    movel([-0.071523, -1.431037, -2.538408, -0.742944, 1.570796, 1.499273],accel_mss,speed_ms,0,blend_radius_m)
    movel([-0.071633, -1.429838, -2.539341, -0.743210, 1.570796, 1.499163],accel_mss,speed_ms,0,blend_radius_m)
    movel([-0.072441, -1.426473, -2.541948, -0.743968, 1.570796, 1.498355],accel_mss,speed_ms,0,blend_radius_m)
    movel([-0.072913, -1.424072, -2.543798, -0.744519, 1.570796, 1.497883],accel_mss,speed_ms,0,blend_radius_m)
    movel([-0.072968, -1.423023, -2.544604, -0.744762, 1.570796, 1.497829],accel_mss,speed_ms,0,blend_radius_m)
    movel([-0.072889, -1.422073, -2.545332, -0.744984, 1.570796, 1.497908],accel_mss,speed_ms,0,blend_radius_m)
    movel([-0.072695, -1.421230, -2.545977, -0.745182, 1.570796, 1.498101],accel_mss,speed_ms,0,blend_radius_m)
    movel([-0.072401, -1.420498, -2.546536, -0.745355, 1.570796, 1.498395],accel_mss,speed_ms,0,blend_radius_m)
    movel([-0.072027, -1.419881, -2.547006, -0.745502, 1.570796, 1.498770],accel_mss,speed_ms,0,blend_radius_m)
    movel([-0.071586, -1.419384, -2.547385, -0.745620, 1.570796, 1.499210],accel_mss,speed_ms,0,blend_radius_m)
    movel([-0.071096, -1.419012, -2.547668, -0.745709, 1.570796, 1.499700],accel_mss,speed_ms,0,blend_radius_m)
    movel([-0.070575, -1.418770, -2.547852, -0.745766, 1.570796, 1.500221],accel_mss,speed_ms,0,blend_radius_m)
    movel([-0.070039, -1.418663, -2.547934, -0.745792, 1.570796, 1.500757],accel_mss,speed_ms,0,blend_radius_m)
    movel([-0.069506, -1.418695, -2.547909, -0.745784, 1.570796, 1.501291],accel_mss,speed_ms,0,blend_radius_m)
    movel([-0.068990, -1.418869, -2.547777, -0.745743, 1.570796, 1.501806],accel_mss,speed_ms,0,blend_radius_m)
    movel([-0.068509, -1.419192, -2.547531, -0.745666, 1.570796, 1.502287],accel_mss,speed_ms,0,blend_radius_m)
    movel([-0.068083, -1.419668, -2.547169, -0.745552, 1.570796, 1.502713],accel_mss,speed_ms,0,blend_radius_m)
    movel([-0.067726, -1.420299, -2.546687, -0.745402, 1.570796, 1.503070],accel_mss,speed_ms,0,blend_radius_m)
    movel([-0.067456, -1.421092, -2.546082, -0.745215, 1.570796, 1.503341],accel_mss,speed_ms,0,blend_radius_m)
    movel([-0.067286, -1.422046, -2.545352, -0.744991, 1.570796, 1.503511],accel_mss,speed_ms,0,blend_radius_m)
    movel([-0.066480, -1.420784, -2.546318, -0.745288, 1.570796, 1.504317],accel_mss,speed_ms,0,blend_radius_m)
    movel([-0.065836, -1.419517, -2.547284, -0.745588, 1.570796, 1.504961],accel_mss,speed_ms,0,blend_radius_m)
    movel([-0.065321, -1.418247, -2.548250, -0.745892, 1.570796, 1.505475],accel_mss,speed_ms,0,blend_radius_m)
    movel([-0.064903, -1.416973, -2.549217, -0.746199, 1.570796, 1.505893],accel_mss,speed_ms,0,blend_radius_m)
    movel([-0.063493, -1.411871, -2.553065, -0.747453, 1.570796, 1.507303],accel_mss,speed_ms,0,blend_radius_m)
    movel([-0.062918, -1.409984, -2.554478, -0.747927, 1.570796, 1.507878],accel_mss,speed_ms,0,blend_radius_m)
    movel([-0.062028, -1.407742, -2.556150, -0.748496, 1.570796, 1.508768],accel_mss,speed_ms,0,blend_radius_m)
    movel([-0.061398, -1.406679, -2.556941, -0.748769, 1.570796, 1.509398],accel_mss,speed_ms,0,blend_radius_m)
    movel([-0.060609, -1.405759, -2.557623, -0.749006, 1.570796, 1.510187],accel_mss,speed_ms,0,blend_radius_m)
    movel([-0.060144, -1.405377, -2.557906, -0.749106, 1.570796, 1.510652],accel_mss,speed_ms,0,blend_radius_m)
    movel([-0.059065, -1.404813, -2.558324, -0.749252, 1.570796, 1.511731],accel_mss,speed_ms,0,blend_radius_m)
    movel([-0.058441, -1.404655, -2.558441, -0.749293, 1.570796, 1.512355],accel_mss,speed_ms,0,blend_radius_m)
    movel([-0.057834, -1.404687, -2.558417, -0.749285, 1.570796, 1.512962],accel_mss,speed_ms,0,blend_radius_m)
    movel([-0.057396, -1.404971, -2.558207, -0.749211, 1.570796, 1.513400],accel_mss,speed_ms,0,blend_radius_m)
    movel([-0.056907, -1.405936, -2.557492, -0.748961, 1.570796, 1.513889],accel_mss,speed_ms,0,blend_radius_m)
    movel([-0.056592, -1.407441, -2.556375, -0.748574, 1.570796, 1.514204],accel_mss,speed_ms,0,blend_radius_m)
    movel([-0.056446, -1.409015, -2.555202, -0.748172, 1.570796, 1.514350],accel_mss,speed_ms,0,blend_radius_m)
    movel([-0.055172, -1.407309, -2.556473, -0.748607, 1.570796, 1.515625],accel_mss,speed_ms,0,blend_radius_m)
    movel([-0.053733, -1.405654, -2.557701, -0.749034, 1.570796, 1.517063],accel_mss,speed_ms,0,blend_radius_m)
    movel([-0.052159, -1.404070, -2.558873, -0.749446, 1.570796, 1.518637],accel_mss,speed_ms,0,blend_radius_m)
    movel([-0.050484, -1.402575, -2.559976, -0.749838, 1.570796, 1.520313],accel_mss,speed_ms,0,blend_radius_m)
    movel([-0.047138, -1.399585, -2.562172, -0.750632, 1.570796, 1.523659],accel_mss,speed_ms,0,blend_radius_m)
    movel([-0.046149, -1.398798, -2.562748, -0.750843, 1.570796, 1.524647],accel_mss,speed_ms,0,blend_radius_m)
    movel([-0.045182, -1.398133, -2.563233, -0.751022, 1.570796, 1.525614],accel_mss,speed_ms,0,blend_radius_m)
    movel([-0.044274, -1.397659, -2.563579, -0.751151, 1.570796, 1.526522],accel_mss,speed_ms,0,blend_radius_m)
    movel([-0.043471, -1.397443, -2.563737, -0.751209, 1.570796, 1.527325],accel_mss,speed_ms,0,blend_radius_m)
    movel([-0.042803, -1.397569, -2.563645, -0.751175, 1.570796, 1.527993],accel_mss,speed_ms,0,blend_radius_m)
    movel([-0.042348, -1.398020, -2.563316, -0.751053, 1.570796, 1.528448],accel_mss,speed_ms,0,blend_radius_m)
    movel([-0.042088, -1.398712, -2.562811, -0.750866, 1.570796, 1.528709],accel_mss,speed_ms,0,blend_radius_m)
    movel([-0.042011, -1.399560, -2.562190, -0.750639, 1.570796, 1.528786],accel_mss,speed_ms,0,blend_radius_m)
    movel([-0.042101, -1.400480, -2.561516, -0.750393, 1.570796, 1.528695],accel_mss,speed_ms,0,blend_radius_m)
    movel([-0.042343, -1.401386, -2.560851, -0.750152, 1.570796, 1.528454],accel_mss,speed_ms,0,blend_radius_m)
    movel([-0.042722, -1.402197, -2.560255, -0.749938, 1.570796, 1.528075],accel_mss,speed_ms,0,blend_radius_m)
    movel([-0.043225, -1.402828, -2.559790, -0.749771, 1.570796, 1.527572],accel_mss,speed_ms,0,blend_radius_m)
    movel([-0.040166, -1.400250, -2.561685, -0.750454, 1.570796, 1.530630],accel_mss,speed_ms,0,blend_radius_m)
    movel([-0.038546, -1.399062, -2.562555, -0.750772, 1.570796, 1.532251],accel_mss,speed_ms,0,blend_radius_m)
    movel([-0.036872, -1.397960, -2.563360, -0.751069, 1.570796, 1.533924],accel_mss,speed_ms,0,blend_radius_m)
    movel([-0.035156, -1.396957, -2.564091, -0.751341, 1.570796, 1.535640],accel_mss,speed_ms,0,blend_radius_m)
    movel([-0.033403, -1.396067, -2.564739, -0.751583, 1.570796, 1.537394],accel_mss,speed_ms,0,blend_radius_m)
    movel([-0.031619, -1.395304, -2.565293, -0.751792, 1.570796, 1.539177],accel_mss,speed_ms,0,blend_radius_m)
    movel([-0.029813, -1.394680, -2.565746, -0.751963, 1.570796, 1.540983],accel_mss,speed_ms,0,blend_radius_m)
    movel([-0.028597, -1.394494, -2.565881, -0.752015, 1.570796, 1.542199],accel_mss,speed_ms,0,blend_radius_m)
    movel([-0.027308, -1.394611, -2.565796, -0.751982, 1.570796, 1.543488],accel_mss,speed_ms,0,blend_radius_m)
    movel([-0.026754, -1.394802, -2.565657, -0.751930, 1.570796, 1.544042],accel_mss,speed_ms,0,blend_radius_m)
    movel([-0.026320, -1.395091, -2.565448, -0.751851, 1.570796, 1.544476],accel_mss,speed_ms,0,blend_radius_m)
    movel([-0.026051, -1.395484, -2.565162, -0.751743, 1.570796, 1.544745],accel_mss,speed_ms,0,blend_radius_m)
    movel([-0.025998, -1.395992, -2.564793, -0.751604, 1.570796, 1.544799],accel_mss,speed_ms,0,blend_radius_m)
    movel([-0.026188, -1.396540, -2.564395, -0.751454, 1.570796, 1.544608],accel_mss,speed_ms,0,blend_radius_m)
    movel([-0.026559, -1.397086, -2.563997, -0.751306, 1.570796, 1.544238],accel_mss,speed_ms,0,blend_radius_m)
    movel([-0.027646, -1.398202, -2.563183, -0.751004, 1.570796, 1.543150],accel_mss,speed_ms,0,blend_radius_m)
    movel([-0.028935, -1.399131, -2.562504, -0.750754, 1.570796, 1.541861],accel_mss,speed_ms,0,blend_radius_m)
    movel([-0.030340, -1.399897, -2.561943, -0.750548, 1.570796, 1.540456],accel_mss,speed_ms,0,blend_radius_m)
    movel([-0.031777, -1.400524, -2.561484, -0.750381, 1.570796, 1.539020],accel_mss,speed_ms,0,blend_radius_m)
    movel([-0.029959, -1.400609, -2.561422, -0.750359, 1.570796, 1.540838],accel_mss,speed_ms,0,blend_radius_m)
    movel([-0.028062, -1.400516, -2.561490, -0.750383, 1.570796, 1.542735],accel_mss,speed_ms,0,blend_radius_m)
    movel([-0.026107, -1.400250, -2.561685, -0.750454, 1.570796, 1.544690],accel_mss,speed_ms,0,blend_radius_m)
    movel([-0.024112, -1.399814, -2.562004, -0.750571, 1.570796, 1.546684],accel_mss,speed_ms,0,blend_radius_m)
    movel([-0.022533, -1.399314, -2.562370, -0.750705, 1.570796, 1.548263],accel_mss,speed_ms,0,blend_radius_m)
    movel([-0.019437, -1.398102, -2.563256, -0.751031, 1.570796, 1.551359],accel_mss,speed_ms,0,blend_radius_m)
    movel([-0.017855, -1.397589, -2.563630, -0.751169, 1.570796, 1.552941],accel_mss,speed_ms,0,blend_radius_m)
    movel([-0.016060, -1.397130, -2.563965, -0.751294, 1.570796, 1.554737],accel_mss,speed_ms,0,blend_radius_m)
    movel([-0.013047, -1.396511, -2.564416, -0.751462, 1.570796, 1.557749],accel_mss,speed_ms,0,blend_radius_m)
    movel([-0.011613, -1.396336, -2.564543, -0.751510, 1.570796, 1.559183],accel_mss,speed_ms,0,blend_radius_m)
    movel([-0.010507, -1.396353, -2.564531, -0.751505, 1.570796, 1.560289],accel_mss,speed_ms,0,blend_radius_m)
    movel([-0.010142, -1.396457, -2.564455, -0.751477, 1.570796, 1.560654],accel_mss,speed_ms,0,blend_radius_m)
    movel([-0.009941, -1.396639, -2.564322, -0.751427, 1.570796, 1.560855],accel_mss,speed_ms,0,blend_radius_m)
    movel([-0.009926, -1.396905, -2.564129, -0.751355, 1.570796, 1.560871],accel_mss,speed_ms,0,blend_radius_m)
    movel([-0.010125, -1.397265, -2.563866, -0.751257, 1.570796, 1.560671],accel_mss,speed_ms,0,blend_radius_m)
    movel([-0.010875, -1.398064, -2.563284, -0.751041, 1.570796, 1.559921],accel_mss,speed_ms,0,blend_radius_m)
    movel([-0.011846, -1.398827, -2.562726, -0.750835, 1.570796, 1.558951],accel_mss,speed_ms,0,blend_radius_m)
    movel([-0.012974, -1.399552, -2.562196, -0.750641, 1.570796, 1.557822],accel_mss,speed_ms,0,blend_radius_m)
    movel([-0.014194, -1.400229, -2.561700, -0.750460, 1.570796, 1.556602],accel_mss,speed_ms,0,blend_radius_m)
    movel([-0.016663, -1.401417, -2.560828, -0.750144, 1.570796, 1.554134],accel_mss,speed_ms,0,blend_radius_m)
    movel([-0.018743, -1.402340, -2.560149, -0.749900, 1.570796, 1.552053],accel_mss,speed_ms,0,blend_radius_m)
    movel([-0.017712, -1.402591, -2.559964, -0.749834, 1.570796, 1.553085],accel_mss,speed_ms,0,blend_radius_m)
    movel([-0.016621, -1.402742, -2.559853, -0.749794, 1.570796, 1.554176],accel_mss,speed_ms,0,blend_radius_m)
    movel([-0.014303, -1.402794, -2.559815, -0.749780, 1.570796, 1.556493],accel_mss,speed_ms,0,blend_radius_m)
    movel([-0.011861, -1.402587, -2.559967, -0.749835, 1.570796, 1.558936],accel_mss,speed_ms,0,blend_radius_m)
    movel([-0.009363, -1.402213, -2.560243, -0.749933, 1.570796, 1.561434],accel_mss,speed_ms,0,blend_radius_m)
    movel([-0.007287, -1.401786, -2.560557, -0.750046, 1.570796, 1.563509],accel_mss,speed_ms,0,blend_radius_m)
    movel([-0.001019, -1.400276, -2.561666, -0.750447, 1.570796, 1.569778],accel_mss,speed_ms,0,blend_radius_m)
    movel([0.000136, -1.400180, -2.561736, -0.750473, 1.570796, 1.570932],accel_mss,speed_ms,0,blend_radius_m)
    movel([0.001035, -1.400358, -2.561606, -0.750426, 1.570796, 1.571832],accel_mss,speed_ms,0,blend_radius_m)
    movel([0.001220, -1.400571, -2.561450, -0.750369, 1.570796, 1.572016],accel_mss,speed_ms,0,blend_radius_m)
    movel([0.001136, -1.400879, -2.561224, -0.750287, 1.570796, 1.571932],accel_mss,speed_ms,0,blend_radius_m)
    movel([0.000714, -1.401289, -2.560922, -0.750178, 1.570796, 1.571510],accel_mss,speed_ms,0,blend_radius_m)
    movel([-0.000113, -1.401810, -2.560539, -0.750040, 1.570796, 1.570683],accel_mss,speed_ms,0,blend_radius_m)
    movel([-0.001501, -1.402493, -2.560036, -0.749859, 1.570796, 1.569296],accel_mss,speed_ms,0,blend_radius_m)
    movel([-0.003103, -1.403126, -2.559570, -0.749693, 1.570796, 1.567693],accel_mss,speed_ms,0,blend_radius_m)
    movel([-0.004684, -1.403568, -2.559244, -0.749577, 1.570796, 1.566113],accel_mss,speed_ms,0,blend_radius_m)
    movel([-0.005392, -1.403675, -2.559165, -0.749549, 1.570796, 1.565405],accel_mss,speed_ms,0,blend_radius_m)
    movel([-0.006002, -1.403679, -2.559162, -0.749548, 1.570796, 1.564794],accel_mss,speed_ms,0,blend_radius_m)
    movel([-0.003636, -1.404544, -2.558523, -0.749322, 1.570796, 1.567160],accel_mss,speed_ms,0,blend_radius_m)
    movel([-0.001096, -1.405162, -2.558066, -0.749161, 1.570796, 1.569700],accel_mss,speed_ms,0,blend_radius_m)
    movel([0.001580, -1.405578, -2.557757, -0.749053, 1.570796, 1.572376],accel_mss,speed_ms,0,blend_radius_m)
    movel([0.004358, -1.405841, -2.557562, -0.748985, 1.570796, 1.575155],accel_mss,speed_ms,0,blend_radius_m)
    movel([0.010072, -1.406085, -2.557382, -0.748922, 1.570796, 1.580868],accel_mss,speed_ms,0,blend_radius_m)
    movel([0.015745, -1.406260, -2.557252, -0.748877, 1.570796, 1.586542],accel_mss,speed_ms,0,blend_radius_m)
    movel([0.016685, -1.406434, -2.557122, -0.748832, 1.570796, 1.587482],accel_mss,speed_ms,0,blend_radius_m)
    movel([0.016994, -1.406671, -2.556947, -0.748771, 1.570796, 1.587790],accel_mss,speed_ms,0,blend_radius_m)
    movel([0.017081, -1.407052, -2.556663, -0.748673, 1.570796, 1.587877],accel_mss,speed_ms,0,blend_radius_m)
    movel([0.016911, -1.407502, -2.556329, -0.748558, 1.570796, 1.587708],accel_mss,speed_ms,0,blend_radius_m)
    movel([0.015985, -1.408575, -2.555530, -0.748284, 1.570796, 1.586781],accel_mss,speed_ms,0,blend_radius_m)
    movel([0.015320, -1.409142, -2.555107, -0.748140, 1.570796, 1.586116],accel_mss,speed_ms,0,blend_radius_m)
    movel([0.013817, -1.410100, -2.554391, -0.747897, 1.570796, 1.584614],accel_mss,speed_ms,0,blend_radius_m)
    movel([0.012159, -1.410835, -2.553841, -0.747712, 1.570796, 1.582955],accel_mss,speed_ms,0,blend_radius_m)
    movel([0.010414, -1.411373, -2.553438, -0.747578, 1.570796, 1.581211],accel_mss,speed_ms,0,blend_radius_m)
    movel([0.008663, -1.411731, -2.553170, -0.747488, 1.570796, 1.579460],accel_mss,speed_ms,0,blend_radius_m)
    movel([0.006980, -1.411932, -2.553019, -0.747438, 1.570796, 1.577776],accel_mss,speed_ms,0,blend_radius_m)
    movel([0.005437, -1.411996, -2.552971, -0.747422, 1.570796, 1.576233],accel_mss,speed_ms,0,blend_radius_m)
    movel([0.004115, -1.411939, -2.553014, -0.747436, 1.570796, 1.574911],accel_mss,speed_ms,0,blend_radius_m)
    movel([0.004101, -1.412306, -2.552739, -0.747345, 1.570796, 1.574897],accel_mss,speed_ms,0,blend_radius_m)
    movel([0.004332, -1.412571, -2.552539, -0.747279, 1.570796, 1.575129],accel_mss,speed_ms,0,blend_radius_m)
    movel([0.005050, -1.413018, -2.552204, -0.747168, 1.570796, 1.575846],accel_mss,speed_ms,0,blend_radius_m)
    movel([0.005864, -1.413355, -2.551950, -0.747084, 1.570796, 1.576660],accel_mss,speed_ms,0,blend_radius_m)
    movel([0.007653, -1.413832, -2.551590, -0.746966, 1.570796, 1.578449],accel_mss,speed_ms,0,blend_radius_m)
    movel([0.010843, -1.414489, -2.551095, -0.746805, 1.570796, 1.581640],accel_mss,speed_ms,0,blend_radius_m)
    movel([0.014087, -1.415030, -2.550687, -0.746672, 1.570796, 1.584883],accel_mss,speed_ms,0,blend_radius_m)
    movel([0.020731, -1.415822, -2.550089, -0.746479, 1.570796, 1.591527],accel_mss,speed_ms,0,blend_radius_m)
    movel([0.022573, -1.416072, -2.549899, -0.746418, 1.570796, 1.593369],accel_mss,speed_ms,0,blend_radius_m)
    movel([0.023740, -1.416328, -2.549705, -0.746355, 1.570796, 1.594536],accel_mss,speed_ms,0,blend_radius_m)
    movel([0.024859, -1.416697, -2.549426, -0.746266, 1.570796, 1.595655],accel_mss,speed_ms,0,blend_radius_m)
    movel([0.025765, -1.417197, -2.549047, -0.746145, 1.570796, 1.596561],accel_mss,speed_ms,0,blend_radius_m)
    movel([0.026296, -1.417842, -2.548558, -0.745989, 1.570796, 1.597093],accel_mss,speed_ms,0,blend_radius_m)
    movel([0.026375, -1.418223, -2.548269, -0.745898, 1.570796, 1.597171],accel_mss,speed_ms,0,blend_radius_m)
    movel([0.026302, -1.418647, -2.547946, -0.745796, 1.570796, 1.597098],accel_mss,speed_ms,0,blend_radius_m)
    movel([0.026053, -1.419117, -2.547588, -0.745684, 1.570796, 1.596850],accel_mss,speed_ms,0,blend_radius_m)
    movel([0.025615, -1.419633, -2.547196, -0.745561, 1.570796, 1.596412],accel_mss,speed_ms,0,blend_radius_m)
    movel([0.024960, -1.420017, -2.546903, -0.745469, 1.570796, 1.595756],accel_mss,speed_ms,0,blend_radius_m)
    movel([0.024058, -1.420281, -2.546701, -0.745407, 1.570796, 1.594855],accel_mss,speed_ms,0,blend_radius_m)
    movel([0.019204, -1.421203, -2.545998, -0.745189, 1.570796, 1.590000],accel_mss,speed_ms,0,blend_radius_m)
    movel([0.017567, -1.421316, -2.545911, -0.745162, 1.570796, 1.588363],accel_mss,speed_ms,0,blend_radius_m)
    movel([0.016862, -1.421258, -2.545955, -0.745176, 1.570796, 1.587658],accel_mss,speed_ms,0,blend_radius_m)
    movel([0.016278, -1.421094, -2.546081, -0.745214, 1.570796, 1.587074],accel_mss,speed_ms,0,blend_radius_m)
    movel([0.018723, -1.422630, -2.544905, -0.744854, 1.570796, 1.589519],accel_mss,speed_ms,0,blend_radius_m)
    movel([0.021438, -1.423860, -2.543961, -0.744568, 1.570796, 1.592234],accel_mss,speed_ms,0,blend_radius_m)
    movel([0.024358, -1.424834, -2.543212, -0.744343, 1.570796, 1.595154],accel_mss,speed_ms,0,blend_radius_m)
    movel([0.027421, -1.425597, -2.542624, -0.744168, 1.570796, 1.598218],accel_mss,speed_ms,0,blend_radius_m)
    movel([0.030058, -1.425902, -2.542389, -0.744098, 1.570796, 1.600854],accel_mss,speed_ms,0,blend_radius_m)
    movel([0.033837, -1.426402, -2.542003, -0.743984, 1.570796, 1.604633],accel_mss,speed_ms,0,blend_radius_m)
    movel([0.035556, -1.426815, -2.541684, -0.743890, 1.570796, 1.606352],accel_mss,speed_ms,0,blend_radius_m)
    movel([0.036847, -1.427381, -2.541247, -0.743762, 1.570796, 1.607643],accel_mss,speed_ms,0,blend_radius_m)
    movel([0.037257, -1.427731, -2.540975, -0.743682, 1.570796, 1.608053],accel_mss,speed_ms,0,blend_radius_m)
    movel([0.037469, -1.428131, -2.540666, -0.743592, 1.570796, 1.608265],accel_mss,speed_ms,0,blend_radius_m)
    movel([0.037455, -1.428587, -2.540312, -0.743490, 1.570796, 1.608252],accel_mss,speed_ms,0,blend_radius_m)
    movel([0.037191, -1.429098, -2.539915, -0.743375, 1.570796, 1.607987],accel_mss,speed_ms,0,blend_radius_m)
    movel([0.036771, -1.429574, -2.539546, -0.743269, 1.570796, 1.607567],accel_mss,speed_ms,0,blend_radius_m)
    movel([0.036278, -1.429998, -2.539217, -0.743174, 1.570796, 1.607075],accel_mss,speed_ms,0,blend_radius_m)
    movel([0.035178, -1.430727, -2.538649, -0.743013, 1.570796, 1.605975],accel_mss,speed_ms,0,blend_radius_m)
    movel([0.033953, -1.431402, -2.538124, -0.742864, 1.570796, 1.604749],accel_mss,speed_ms,0,blend_radius_m)
    movel([0.031448, -1.432496, -2.537270, -0.742624, 1.570796, 1.602244],accel_mss,speed_ms,0,blend_radius_m)
    movel([0.030184, -1.432911, -2.536945, -0.742533, 1.570796, 1.600981],accel_mss,speed_ms,0,blend_radius_m)
    movel([0.032542, -1.433431, -2.536538, -0.742420, 1.570796, 1.603338],accel_mss,speed_ms,0,blend_radius_m)
    movel([0.034969, -1.433808, -2.536243, -0.742338, 1.570796, 1.605765],accel_mss,speed_ms,0,blend_radius_m)
    movel([0.037457, -1.434060, -2.536045, -0.742284, 1.570796, 1.608253],accel_mss,speed_ms,0,blend_radius_m)
    movel([0.040000, -1.434199, -2.535936, -0.742253, 1.570796, 1.610797],accel_mss,speed_ms,0,blend_radius_m)
    movel([0.045221, -1.434207, -2.535930, -0.742252, 1.570796, 1.616017],accel_mss,speed_ms,0,blend_radius_m)
    movel([0.050575, -1.433945, -2.536136, -0.742309, 1.570796, 1.621371],accel_mss,speed_ms,0,blend_radius_m)
    movel([0.051984, -1.434006, -2.536088, -0.742295, 1.570796, 1.622781],accel_mss,speed_ms,0,blend_radius_m)
    movel([0.052501, -1.434244, -2.535901, -0.742244, 1.570796, 1.623297],accel_mss,speed_ms,0,blend_radius_m)
    movel([0.052736, -1.434706, -2.535539, -0.742144, 1.570796, 1.623532],accel_mss,speed_ms,0,blend_radius_m)
    movel([0.052700, -1.435095, -2.535234, -0.742061, 1.570796, 1.623496],accel_mss,speed_ms,0,blend_radius_m)
    movel([0.052533, -1.435492, -2.534921, -0.741975, 1.570796, 1.623330],accel_mss,speed_ms,0,blend_radius_m)
    movel([0.051867, -1.436310, -2.534278, -0.741801, 1.570796, 1.622663],accel_mss,speed_ms,0,blend_radius_m)
    movel([0.050864, -1.437120, -2.533640, -0.741629, 1.570796, 1.621660],accel_mss,speed_ms,0,blend_radius_m)
    movel([0.049650, -1.437891, -2.533032, -0.741467, 1.570796, 1.620446],accel_mss,speed_ms,0,blend_radius_m)
    movel([0.047098, -1.439176, -2.532015, -0.741197, 1.570796, 1.617895],accel_mss,speed_ms,0,blend_radius_m)
    movel([0.045218, -1.439885, -2.531454, -0.741050, 1.570796, 1.616015],accel_mss,speed_ms,0,blend_radius_m)
    movel([0.046303, -1.439936, -2.531413, -0.741039, 1.570796, 1.617099],accel_mss,speed_ms,0,blend_radius_m)
    movel([0.047423, -1.439889, -2.531451, -0.741049, 1.570796, 1.618219],accel_mss,speed_ms,0,blend_radius_m)
    movel([0.049742, -1.439530, -2.531735, -0.741124, 1.570796, 1.620538],accel_mss,speed_ms,0,blend_radius_m)
    movel([0.052127, -1.438842, -2.532280, -0.741267, 1.570796, 1.622924],accel_mss,speed_ms,0,blend_radius_m)
    movel([0.054533, -1.437867, -2.533050, -0.741472, 1.570796, 1.625330],accel_mss,speed_ms,0,blend_radius_m)
    movel([0.056914, -1.436636, -2.534021, -0.741732, 1.570796, 1.627711],accel_mss,speed_ms,0,blend_radius_m)
    movel([0.059223, -1.435192, -2.535157, -0.742040, 1.570796, 1.630019],accel_mss,speed_ms,0,blend_radius_m)
    movel([0.061412, -1.433566, -2.536433, -0.742391, 1.570796, 1.632208],accel_mss,speed_ms,0,blend_radius_m)
    movel([0.063435, -1.431798, -2.537814, -0.742777, 1.570796, 1.634231],accel_mss,speed_ms,0,blend_radius_m)
    movel([0.064325, -1.431007, -2.538431, -0.742951, 1.570796, 1.635121],accel_mss,speed_ms,0,blend_radius_m)
    movel([0.064810, -1.430692, -2.538676, -0.743020, 1.570796, 1.635607],accel_mss,speed_ms,0,blend_radius_m)
    movel([0.065322, -1.430491, -2.538833, -0.743065, 1.570796, 1.636119],accel_mss,speed_ms,0,blend_radius_m)
    movel([0.065860, -1.430459, -2.538858, -0.743072, 1.570796, 1.636657],accel_mss,speed_ms,0,blend_radius_m)
    movel([0.066324, -1.430583, -2.538762, -0.743045, 1.570796, 1.637120],accel_mss,speed_ms,0,blend_radius_m)
    movel([0.066842, -1.431005, -2.538433, -0.742951, 1.570796, 1.637638],accel_mss,speed_ms,0,blend_radius_m)
    movel([0.067132, -1.431666, -2.537918, -0.742806, 1.570796, 1.637928],accel_mss,speed_ms,0,blend_radius_m)
    movel([0.067232, -1.432498, -2.537267, -0.742623, 1.570796, 1.638028],accel_mss,speed_ms,0,blend_radius_m)
    movel([0.067182, -1.433445, -2.536527, -0.742417, 1.570796, 1.637978],accel_mss,speed_ms,0,blend_radius_m)
    movel([0.066780, -1.435417, -2.534981, -0.741992, 1.570796, 1.637576],accel_mss,speed_ms,0,blend_radius_m)
    movel([0.066238, -1.437082, -2.533670, -0.741637, 1.570796, 1.637035],accel_mss,speed_ms,0,blend_radius_m)
    movel([0.067950, -1.435277, -2.535090, -0.742022, 1.570796, 1.638746],accel_mss,speed_ms,0,blend_radius_m)
    movel([0.069463, -1.433379, -2.536579, -0.742431, 1.570796, 1.640260],accel_mss,speed_ms,0,blend_radius_m)
    movel([0.070769, -1.431410, -2.538117, -0.742862, 1.570796, 1.641565],accel_mss,speed_ms,0,blend_radius_m)
    movel([0.071860, -1.429398, -2.539683, -0.743308, 1.570796, 1.642657],accel_mss,speed_ms,0,blend_radius_m)
    movel([0.072723, -1.427369, -2.541256, -0.743764, 1.570796, 1.643520],accel_mss,speed_ms,0,blend_radius_m)
    movel([0.073356, -1.425347, -2.542817, -0.744225, 1.570796, 1.644153],accel_mss,speed_ms,0,blend_radius_m)
    movel([0.073744, -1.423362, -2.544343, -0.744683, 1.570796, 1.644540],accel_mss,speed_ms,0,blend_radius_m)
    movel([0.073879, -1.421440, -2.545816, -0.745133, 1.570796, 1.644675],accel_mss,speed_ms,0,blend_radius_m)
    movel([0.073661, -1.418892, -2.547760, -0.745737, 1.570796, 1.644458],accel_mss,speed_ms,0,blend_radius_m)
    movel([0.073663, -1.417520, -2.548802, -0.746067, 1.570796, 1.644460],accel_mss,speed_ms,0,blend_radius_m)
    movel([0.073776, -1.416854, -2.549307, -0.746228, 1.570796, 1.644572],accel_mss,speed_ms,0,blend_radius_m)
    movel([0.073991, -1.416217, -2.549790, -0.746382, 1.570796, 1.644787],accel_mss,speed_ms,0,blend_radius_m)
    movel([0.074550, -1.415234, -2.550533, -0.746622, 1.570796, 1.645347],accel_mss,speed_ms,0,blend_radius_m)
    movel([0.075106, -1.414698, -2.550937, -0.746753, 1.570796, 1.645903],accel_mss,speed_ms,0,blend_radius_m)
    movel([0.075657, -1.414513, -2.551077, -0.746799, 1.570796, 1.646454],accel_mss,speed_ms,0,blend_radius_m)
    movel([0.076198, -1.414581, -2.551026, -0.746782, 1.570796, 1.646994],accel_mss,speed_ms,0,blend_radius_m)
    movel([0.077684, -1.415340, -2.550453, -0.746596, 1.570796, 1.648480],accel_mss,speed_ms,0,blend_radius_m)
    movel([0.078118, -1.415453, -2.550367, -0.746569, 1.570796, 1.648914],accel_mss,speed_ms,0,blend_radius_m)
    movel([0.078894, -1.413988, -2.551473, -0.746928, 1.570796, 1.649690],accel_mss,speed_ms,0,blend_radius_m)
    movel([0.079523, -1.412498, -2.552594, -0.747297, 1.570796, 1.650319],accel_mss,speed_ms,0,blend_radius_m)
    movel([0.080014, -1.410991, -2.553724, -0.747673, 1.570796, 1.650810],accel_mss,speed_ms,0,blend_radius_m)
    movel([0.080375, -1.409474, -2.554859, -0.748056, 1.570796, 1.651171],accel_mss,speed_ms,0,blend_radius_m)
    movel([0.080608, -1.407958, -2.555990, -0.748441, 1.570796, 1.651405],accel_mss,speed_ms,0,blend_radius_m)
    movel([0.080723, -1.406448, -2.557113, -0.748829, 1.570796, 1.651520],accel_mss,speed_ms,0,blend_radius_m)
    movel([0.080635, -1.403476, -2.559312, -0.749601, 1.570796, 1.651431],accel_mss,speed_ms,0,blend_radius_m)
    movel([0.080162, -1.400629, -2.561407, -0.750353, 1.570796, 1.650958],accel_mss,speed_ms,0,blend_radius_m)
    movel([0.079372, -1.397967, -2.563355, -0.751067, 1.570796, 1.650169],accel_mss,speed_ms,0,blend_radius_m)
    movel([0.078320, -1.395559, -2.565108, -0.751722, 1.570796, 1.649116],accel_mss,speed_ms,0,blend_radius_m)
    movel([0.077075, -1.393466, -2.566625, -0.752298, 1.570796, 1.647871],accel_mss,speed_ms,0,blend_radius_m)
    speed_ms = 0.005
    movel([0.077075, -1.384778, -2.562689, -0.764923, 1.570796, 1.647871],accel_mss,speed_ms,0,blend_radius_m)
    speed_ms = 0.040
    movel([0.063534, -1.389965, -2.558967, -0.763456, 1.570796, 1.634331],accel_mss,speed_ms,0,blend_radius_m)
    speed_ms = 0.005
    movel([0.063534, -1.398616, -2.562881, -0.750892, 1.570796, 1.634331],accel_mss,speed_ms,0,blend_radius_m)
    speed_ms = 0.025
    movel([0.062308, -1.398046, -2.563297, -0.751046, 1.570796, 1.633105],accel_mss,speed_ms,0,blend_radius_m)
    movel([0.060907, -1.397768, -2.563500, -0.751121, 1.570796, 1.631703],accel_mss,speed_ms,0,blend_radius_m)
    movel([0.059365, -1.397742, -2.563519, -0.751128, 1.570796, 1.630162],accel_mss,speed_ms,0,blend_radius_m)
    movel([0.057724, -1.397927, -2.563384, -0.751078, 1.570796, 1.628520],accel_mss,speed_ms,0,blend_radius_m)
    movel([0.056020, -1.398282, -2.563124, -0.750982, 1.570796, 1.626816],accel_mss,speed_ms,0,blend_radius_m)
    movel([0.054289, -1.398767, -2.562771, -0.750852, 1.570796, 1.625085],accel_mss,speed_ms,0,blend_radius_m)
    movel([0.050898, -1.399957, -2.561899, -0.750532, 1.570796, 1.621694],accel_mss,speed_ms,0,blend_radius_m)
    speed_ms = 0.005
    movel([0.050898, -1.391317, -2.557992, -0.763081, 1.570796, 1.621694],accel_mss,speed_ms,0,blend_radius_m)
    speed_ms = 0.040
    movel([0.055256, -1.389402, -2.559373, -0.763614, 1.570796, 1.626053],accel_mss,speed_ms,0,blend_radius_m)
    speed_ms = 0.005
    movel([0.055256, -1.398057, -2.563289, -0.751043, 1.570796, 1.626053],accel_mss,speed_ms,0,blend_radius_m)
    speed_ms = 0.025
    movel([0.055845, -1.396352, -2.564531, -0.751505, 1.570796, 1.626642],accel_mss,speed_ms,0,blend_radius_m)
    movel([0.056245, -1.394719, -2.565717, -0.751953, 1.570796, 1.627041],accel_mss,speed_ms,0,blend_radius_m)
    movel([0.056459, -1.393154, -2.566850, -0.752385, 1.570796, 1.627255],accel_mss,speed_ms,0,blend_radius_m)
    movel([0.056496, -1.391653, -2.567934, -0.752803, 1.570796, 1.627292],accel_mss,speed_ms,0,blend_radius_m)
    movel([0.056368, -1.390210, -2.568972, -0.753207, 1.570796, 1.627164],accel_mss,speed_ms,0,blend_radius_m)
    movel([0.056082, -1.388822, -2.569967, -0.753599, 1.570796, 1.626878],accel_mss,speed_ms,0,blend_radius_m)
    movel([0.055647, -1.387485, -2.570924, -0.753980, 1.570796, 1.626443],accel_mss,speed_ms,0,blend_radius_m)
    movel([0.055072, -1.386194, -2.571845, -0.754350, 1.570796, 1.625868],accel_mss,speed_ms,0,blend_radius_m)
    movel([0.052987, -1.382648, -2.574363, -0.755378, 1.570796, 1.623783],accel_mss,speed_ms,0,blend_radius_m)
    movel([0.052074, -1.380895, -2.575601, -0.755893, 1.570796, 1.622870],accel_mss,speed_ms,0,blend_radius_m)
    movel([0.051383, -1.378804, -2.577072, -0.756513, 1.570796, 1.622179],accel_mss,speed_ms,0,blend_radius_m)
    movel([0.050854, -1.376012, -2.579026, -0.757351, 1.570796, 1.621650],accel_mss,speed_ms,0,blend_radius_m)
    movel([0.050603, -1.373085, -2.581063, -0.758241, 1.570796, 1.621400],accel_mss,speed_ms,0,blend_radius_m)
    movel([0.050727, -1.370017, -2.583184, -0.759188, 1.570796, 1.621523],accel_mss,speed_ms,0,blend_radius_m)
    movel([0.050958, -1.368427, -2.584278, -0.759683, 1.570796, 1.621754],accel_mss,speed_ms,0,blend_radius_m)
    movel([0.051319, -1.366802, -2.585393, -0.760194, 1.570796, 1.622116],accel_mss,speed_ms,0,blend_radius_m)
    movel([0.052166, -1.364265, -2.587126, -0.760998, 1.570796, 1.622963],accel_mss,speed_ms,0,blend_radius_m)
    movel([0.053347, -1.361793, -2.588805, -0.761790, 1.570796, 1.624143],accel_mss,speed_ms,0,blend_radius_m)
    movel([0.054842, -1.359405, -2.590420, -0.762564, 1.570796, 1.625638],accel_mss,speed_ms,0,blend_radius_m)
    movel([0.056631, -1.357118, -2.591958, -0.763313, 1.570796, 1.627428],accel_mss,speed_ms,0,blend_radius_m)
    movel([0.058692, -1.354955, -2.593406, -0.764027, 1.570796, 1.629488],accel_mss,speed_ms,0,blend_radius_m)
    movel([0.061006, -1.352938, -2.594751, -0.764700, 1.570796, 1.631802],accel_mss,speed_ms,0,blend_radius_m)
    movel([0.063550, -1.351083, -2.595983, -0.765323, 1.570796, 1.634346],accel_mss,speed_ms,0,blend_radius_m)
    movel([0.066300, -1.349415, -2.597086, -0.765888, 1.570796, 1.637096],accel_mss,speed_ms,0,blend_radius_m)
    movel([0.068452, -1.348320, -2.597808, -0.766261, 1.570796, 1.639248],accel_mss,speed_ms,0,blend_radius_m)
    movel([0.070649, -1.347377, -2.598429, -0.766583, 1.570796, 1.641446],accel_mss,speed_ms,0,blend_radius_m)
    movel([0.072869, -1.346592, -2.598945, -0.766852, 1.570796, 1.643665],accel_mss,speed_ms,0,blend_radius_m)
    movel([0.075095, -1.345963, -2.599358, -0.767069, 1.570796, 1.645892],accel_mss,speed_ms,0,blend_radius_m)
    movel([0.077306, -1.345498, -2.599662, -0.767229, 1.570796, 1.648102],accel_mss,speed_ms,0,blend_radius_m)
    movel([0.079481, -1.345198, -2.599858, -0.767332, 1.570796, 1.650277],accel_mss,speed_ms,0,blend_radius_m)
    movel([0.081599, -1.345066, -2.599945, -0.767378, 1.570796, 1.652396],accel_mss,speed_ms,0,blend_radius_m)
    movel([0.083642, -1.345105, -2.599920, -0.767365, 1.570796, 1.654438],accel_mss,speed_ms,0,blend_radius_m)
    movel([0.085586, -1.345316, -2.599781, -0.767292, 1.570796, 1.656383],accel_mss,speed_ms,0,blend_radius_m)
    movel([0.087417, -1.345701, -2.599529, -0.767159, 1.570796, 1.658213],accel_mss,speed_ms,0,blend_radius_m)
    movel([0.089112, -1.346262, -2.599161, -0.766966, 1.570796, 1.659909],accel_mss,speed_ms,0,blend_radius_m)
    movel([0.090654, -1.347000, -2.598677, -0.766712, 1.570796, 1.661451],accel_mss,speed_ms,0,blend_radius_m)
    movel([0.092024, -1.347915, -2.598075, -0.766399, 1.570796, 1.662821],accel_mss,speed_ms,0,blend_radius_m)
    movel([0.093200, -1.349010, -2.597353, -0.766025, 1.570796, 1.663996],accel_mss,speed_ms,0,blend_radius_m)
    movel([0.094165, -1.350283, -2.596513, -0.765594, 1.570796, 1.664962],accel_mss,speed_ms,0,blend_radius_m)
    movel([0.094904, -1.351735, -2.595550, -0.765103, 1.570796, 1.665700],accel_mss,speed_ms,0,blend_radius_m)
    movel([0.095574, -1.353804, -2.594175, -0.764411, 1.570796, 1.666370],accel_mss,speed_ms,0,blend_radius_m)
    movel([0.096022, -1.355987, -2.592716, -0.763686, 1.570796, 1.666818],accel_mss,speed_ms,0,blend_radius_m)
    movel([0.096290, -1.358256, -2.591193, -0.762939, 1.570796, 1.667086],accel_mss,speed_ms,0,blend_radius_m)
    movel([0.096428, -1.360573, -2.589631, -0.762185, 1.570796, 1.667225],accel_mss,speed_ms,0,blend_radius_m)
    movel([0.096459, -1.365683, -2.586158, -0.760547, 1.570796, 1.667255],accel_mss,speed_ms,0,blend_radius_m)
    movel([0.096218, -1.370867, -2.582598, -0.758924, 1.570796, 1.667014],accel_mss,speed_ms,0,blend_radius_m)
    movel([0.095765, -1.376098, -2.578966, -0.757325, 1.570796, 1.666561],accel_mss,speed_ms,0,blend_radius_m)
    movel([0.095158, -1.381344, -2.575284, -0.755761, 1.570796, 1.665954],accel_mss,speed_ms,0,blend_radius_m)
    movel([0.092366, -1.401990, -2.560407, -0.749992, 1.570796, 1.663163],accel_mss,speed_ms,0,blend_radius_m)
    movel([0.091335, -1.411938, -2.553014, -0.747436, 1.570796, 1.662131],accel_mss,speed_ms,0,blend_radius_m)
    movel([0.090990, -1.416821, -2.549332, -0.746236, 1.570796, 1.661787],accel_mss,speed_ms,0,blend_radius_m)
    movel([0.090816, -1.421612, -2.545684, -0.745092, 1.570796, 1.661612],accel_mss,speed_ms,0,blend_radius_m)
    movel([0.090850, -1.426299, -2.542083, -0.744007, 1.570796, 1.661646],accel_mss,speed_ms,0,blend_radius_m)
    movel([0.091133, -1.430860, -2.538546, -0.742983, 1.570796, 1.661929],accel_mss,speed_ms,0,blend_radius_m)
    movel([0.091699, -1.435282, -2.535086, -0.742020, 1.570796, 1.662496],accel_mss,speed_ms,0,blend_radius_m)
    movel([0.092592, -1.439548, -2.531721, -0.741120, 1.570796, 1.663389],accel_mss,speed_ms,0,blend_radius_m)
    movel([0.093072, -1.441144, -2.530455, -0.740790, 1.570796, 1.663868],accel_mss,speed_ms,0,blend_radius_m)
    movel([0.093769, -1.442611, -2.529287, -0.740490, 1.570796, 1.664566],accel_mss,speed_ms,0,blend_radius_m)
    movel([0.094791, -1.443803, -2.528336, -0.740249, 1.570796, 1.665587],accel_mss,speed_ms,0,blend_radius_m)
    movel([0.095458, -1.444250, -2.527979, -0.740160, 1.570796, 1.666254],accel_mss,speed_ms,0,blend_radius_m)
    movel([0.096248, -1.444571, -2.527722, -0.740095, 1.570796, 1.667044],accel_mss,speed_ms,0,blend_radius_m)
    speed_ms = 0.005
    movel([0.096248, -1.436269, -2.524005, -0.752114, 1.570796, 1.667044],accel_mss,speed_ms,0,blend_radius_m)
    speed_ms = 0.040
    movel([0.078916, -1.416288, -2.539481, -0.756620, 1.570796, 1.649712],accel_mss,speed_ms,0,blend_radius_m)
    speed_ms = 0.005
    movel([0.078916, -1.424743, -2.543282, -0.744364, 1.570796, 1.649712],accel_mss,speed_ms,0,blend_radius_m)
    speed_ms = 0.025
    movel([0.078412, -1.425357, -2.542809, -0.744223, 1.570796, 1.649209],accel_mss,speed_ms,0,blend_radius_m)
    movel([0.078051, -1.426030, -2.542290, -0.744069, 1.570796, 1.648847],accel_mss,speed_ms,0,blend_radius_m)
    movel([0.077820, -1.426746, -2.541737, -0.743906, 1.570796, 1.648616],accel_mss,speed_ms,0,blend_radius_m)
    movel([0.077697, -1.427504, -2.541151, -0.743734, 1.570796, 1.648493],accel_mss,speed_ms,0,blend_radius_m)
    movel([0.077723, -1.429102, -2.539913, -0.743374, 1.570796, 1.648520],accel_mss,speed_ms,0,blend_radius_m)
    movel([0.078001, -1.430754, -2.538628, -0.743007, 1.570796, 1.648797],accel_mss,speed_ms,0,blend_radius_m)
    movel([0.079082, -1.435370, -2.535018, -0.742002, 1.570796, 1.649878],accel_mss,speed_ms,0,blend_radius_m)
    movel([0.079104, -1.436572, -2.534072, -0.741745, 1.570796, 1.649901],accel_mss,speed_ms,0,blend_radius_m)
    movel([0.078916, -1.437115, -2.533644, -0.741630, 1.570796, 1.649712],accel_mss,speed_ms,0,blend_radius_m)
    movel([0.078535, -1.437519, -2.533325, -0.741545, 1.570796, 1.649331],accel_mss,speed_ms,0,blend_radius_m)
    movel([0.078154, -1.437719, -2.533168, -0.741503, 1.570796, 1.648951],accel_mss,speed_ms,0,blend_radius_m)
    movel([0.077777, -1.437738, -2.533152, -0.741499, 1.570796, 1.648573],accel_mss,speed_ms,0,blend_radius_m)
    movel([0.077405, -1.437603, -2.533259, -0.741527, 1.570796, 1.648201],accel_mss,speed_ms,0,blend_radius_m)
    movel([0.076691, -1.436956, -2.533769, -0.741664, 1.570796, 1.647488],accel_mss,speed_ms,0,blend_radius_m)
    movel([0.076042, -1.435967, -2.534548, -0.741874, 1.570796, 1.646839],accel_mss,speed_ms,0,blend_radius_m)
    movel([0.075042, -1.433714, -2.536316, -0.742359, 1.570796, 1.645838],accel_mss,speed_ms,0,blend_radius_m)
    movel([0.074639, -1.432352, -2.537382, -0.742655, 1.570796, 1.645436],accel_mss,speed_ms,0,blend_radius_m)
    movel([0.074053, -1.434423, -2.535761, -0.742205, 1.570796, 1.644850],accel_mss,speed_ms,0,blend_radius_m)
    movel([0.073791, -1.436439, -2.534176, -0.741774, 1.570796, 1.644588],accel_mss,speed_ms,0,blend_radius_m)
    movel([0.073806, -1.438397, -2.532632, -0.741360, 1.570796, 1.644602],accel_mss,speed_ms,0,blend_radius_m)
    movel([0.074054, -1.440284, -2.531138, -0.740967, 1.570796, 1.644850],accel_mss,speed_ms,0,blend_radius_m)
    movel([0.074488, -1.442098, -2.529696, -0.740595, 1.570796, 1.645284],accel_mss,speed_ms,0,blend_radius_m)
    movel([0.075067, -1.443826, -2.528318, -0.740245, 1.570796, 1.645864],accel_mss,speed_ms,0,blend_radius_m)
    movel([0.076478, -1.447000, -2.525775, -0.739614, 1.570796, 1.647274],accel_mss,speed_ms,0,blend_radius_m)
    movel([0.076576, -1.447692, -2.525219, -0.739478, 1.570796, 1.647372],accel_mss,speed_ms,0,blend_radius_m)
    movel([0.076429, -1.448031, -2.524946, -0.739412, 1.570796, 1.647226],accel_mss,speed_ms,0,blend_radius_m)
    movel([0.076109, -1.448265, -2.524757, -0.739366, 1.570796, 1.646906],accel_mss,speed_ms,0,blend_radius_m)
    movel([0.075674, -1.448302, -2.524728, -0.739359, 1.570796, 1.646470],accel_mss,speed_ms,0,blend_radius_m)
    movel([0.074709, -1.448109, -2.524884, -0.739397, 1.570796, 1.645505],accel_mss,speed_ms,0,blend_radius_m)
    movel([0.073883, -1.447747, -2.525175, -0.739467, 1.570796, 1.644679],accel_mss,speed_ms,0,blend_radius_m)
    movel([0.073179, -1.447243, -2.525580, -0.739566, 1.570796, 1.643975],accel_mss,speed_ms,0,blend_radius_m)
    movel([0.072589, -1.446616, -2.526084, -0.739689, 1.570796, 1.643385],accel_mss,speed_ms,0,blend_radius_m)
    movel([0.071703, -1.445100, -2.527299, -0.739989, 1.570796, 1.642499],accel_mss,speed_ms,0,blend_radius_m)
    movel([0.071134, -1.443390, -2.528666, -0.740333, 1.570796, 1.641930],accel_mss,speed_ms,0,blend_radius_m)
    movel([0.071098, -1.446951, -2.525815, -0.739623, 1.570796, 1.641895],accel_mss,speed_ms,0,blend_radius_m)
    movel([0.071279, -1.448639, -2.524456, -0.739294, 1.570796, 1.642076],accel_mss,speed_ms,0,blend_radius_m)
    movel([0.071710, -1.450227, -2.523174, -0.738988, 1.570796, 1.642506],accel_mss,speed_ms,0,blend_radius_m)
    movel([0.072398, -1.451443, -2.522190, -0.738756, 1.570796, 1.643195],accel_mss,speed_ms,0,blend_radius_m)
    movel([0.074140, -1.453486, -2.520531, -0.738372, 1.570796, 1.644936],accel_mss,speed_ms,0,blend_radius_m)
    movel([0.074785, -1.454677, -2.519561, -0.738151, 1.570796, 1.645582],accel_mss,speed_ms,0,blend_radius_m)
    movel([0.074853, -1.454950, -2.519339, -0.738101, 1.570796, 1.645650],accel_mss,speed_ms,0,blend_radius_m)
    movel([0.074790, -1.455254, -2.519090, -0.738045, 1.570796, 1.645587],accel_mss,speed_ms,0,blend_radius_m)
    movel([0.074515, -1.455524, -2.518870, -0.737995, 1.570796, 1.645311],accel_mss,speed_ms,0,blend_radius_m)
    movel([0.074033, -1.455724, -2.518706, -0.737958, 1.570796, 1.644829],accel_mss,speed_ms,0,blend_radius_m)
    movel([0.072714, -1.455964, -2.518510, -0.737915, 1.570796, 1.643511],accel_mss,speed_ms,0,blend_radius_m)
    movel([0.070510, -1.456061, -2.518431, -0.737897, 1.570796, 1.641307],accel_mss,speed_ms,0,blend_radius_m)
    movel([0.070864, -1.457061, -2.517613, -0.737715, 1.570796, 1.641660],accel_mss,speed_ms,0,blend_radius_m)
    movel([0.071388, -1.458170, -2.516703, -0.737515, 1.570796, 1.642184],accel_mss,speed_ms,0,blend_radius_m)
    movel([0.072126, -1.459328, -2.515752, -0.737309, 1.570796, 1.642922],accel_mss,speed_ms,0,blend_radius_m)
    movel([0.073121, -1.460476, -2.514807, -0.737106, 1.570796, 1.643918],accel_mss,speed_ms,0,blend_radius_m)
    movel([0.075908, -1.462059, -2.513500, -0.736830, 1.570796, 1.646704],accel_mss,speed_ms,0,blend_radius_m)
    movel([0.077452, -1.462999, -2.512722, -0.736668, 1.570796, 1.648248],accel_mss,speed_ms,0,blend_radius_m)
    movel([0.077903, -1.463405, -2.512386, -0.736599, 1.570796, 1.648700],accel_mss,speed_ms,0,blend_radius_m)
    movel([0.078007, -1.463729, -2.512117, -0.736543, 1.570796, 1.648803],accel_mss,speed_ms,0,blend_radius_m)
    movel([0.077818, -1.464034, -2.511864, -0.736491, 1.570796, 1.648615],accel_mss,speed_ms,0,blend_radius_m)
    movel([0.077530, -1.464298, -2.511645, -0.736446, 1.570796, 1.648326],accel_mss,speed_ms,0,blend_radius_m)
    movel([0.076815, -1.464637, -2.511363, -0.736389, 1.570796, 1.647612],accel_mss,speed_ms,0,blend_radius_m)
    movel([0.076216, -1.464716, -2.511298, -0.736376, 1.570796, 1.647012],accel_mss,speed_ms,0,blend_radius_m)
    movel([0.075614, -1.464692, -2.511317, -0.736380, 1.570796, 1.646411],accel_mss,speed_ms,0,blend_radius_m)
    movel([0.074473, -1.464567, -2.511422, -0.736401, 1.570796, 1.645270],accel_mss,speed_ms,0,blend_radius_m)
    movel([0.075009, -1.465923, -2.510294, -0.736173, 1.570796, 1.645806],accel_mss,speed_ms,0,blend_radius_m)
    movel([0.075674, -1.467200, -2.509228, -0.735961, 1.570796, 1.646470],accel_mss,speed_ms,0,blend_radius_m)
    movel([0.076466, -1.468393, -2.508231, -0.735765, 1.570796, 1.647262],accel_mss,speed_ms,0,blend_radius_m)
    movel([0.077373, -1.469499, -2.507305, -0.735585, 1.570796, 1.648169],accel_mss,speed_ms,0,blend_radius_m)
    movel([0.078449, -1.470443, -2.506513, -0.735433, 1.570796, 1.649245],accel_mss,speed_ms,0,blend_radius_m)
    movel([0.079711, -1.471207, -2.505871, -0.735311, 1.570796, 1.650507],accel_mss,speed_ms,0,blend_radius_m)
    movel([0.082476, -1.472464, -2.504812, -0.735113, 1.570796, 1.653272],accel_mss,speed_ms,0,blend_radius_m)
    movel([0.083182, -1.472936, -2.504414, -0.735039, 1.570796, 1.653978],accel_mss,speed_ms,0,blend_radius_m)
    movel([0.083345, -1.473281, -2.504123, -0.734985, 1.570796, 1.654141],accel_mss,speed_ms,0,blend_radius_m)
    movel([0.083265, -1.473705, -2.503765, -0.734919, 1.570796, 1.654062],accel_mss,speed_ms,0,blend_radius_m)
    movel([0.082989, -1.474068, -2.503458, -0.734863, 1.570796, 1.653785],accel_mss,speed_ms,0,blend_radius_m)
    movel([0.082593, -1.474354, -2.503216, -0.734819, 1.570796, 1.653389],accel_mss,speed_ms,0,blend_radius_m)
    movel([0.081656, -1.474731, -2.502897, -0.734761, 1.570796, 1.652452],accel_mss,speed_ms,0,blend_radius_m)
    movel([0.080412, -1.475013, -2.502658, -0.734718, 1.570796, 1.651208],accel_mss,speed_ms,0,blend_radius_m)
    movel([0.079209, -1.475159, -2.502535, -0.734695, 1.570796, 1.650005],accel_mss,speed_ms,0,blend_radius_m)
    movel([0.078043, -1.475189, -2.502509, -0.734691, 1.570796, 1.648840],accel_mss,speed_ms,0,blend_radius_m)
    movel([0.076913, -1.475118, -2.502569, -0.734702, 1.570796, 1.647709],accel_mss,speed_ms,0,blend_radius_m)
    movel([0.077649, -1.476142, -2.501701, -0.734546, 1.570796, 1.648445],accel_mss,speed_ms,0,blend_radius_m)
    movel([0.078529, -1.477041, -2.500937, -0.734411, 1.570796, 1.649325],accel_mss,speed_ms,0,blend_radius_m)
    movel([0.079550, -1.477797, -2.500294, -0.734298, 1.570796, 1.650346],accel_mss,speed_ms,0,blend_radius_m)
    movel([0.080706, -1.478392, -2.499787, -0.734210, 1.570796, 1.651502],accel_mss,speed_ms,0,blend_radius_m)
    movel([0.081997, -1.478807, -2.499433, -0.734149, 1.570796, 1.652793],accel_mss,speed_ms,0,blend_radius_m)
    movel([0.083421, -1.479026, -2.499246, -0.734116, 1.570796, 1.654217],accel_mss,speed_ms,0,blend_radius_m)
    movel([0.084975, -1.479027, -2.499245, -0.734116, 1.570796, 1.655771],accel_mss,speed_ms,0,blend_radius_m)
    movel([0.086658, -1.478795, -2.499443, -0.734150, 1.570796, 1.657454],accel_mss,speed_ms,0,blend_radius_m)
    speed_ms = 0.005
    movel([0.086658, -1.470763, -2.495867, -0.745759, 1.570796, 1.657454],accel_mss,speed_ms,0,blend_radius_m)
    speed_ms = 0.040
    movel([0.093371, -1.462726, -2.502586, -0.747077, 1.570796, 1.664167],accel_mss,speed_ms,0,blend_radius_m)
    speed_ms = 0.005
    movel([0.093371, -1.470822, -2.506195, -0.735373, 1.570796, 1.664167],accel_mss,speed_ms,0,blend_radius_m)
    speed_ms = 0.025
    movel([0.090188, -1.470014, -2.506873, -0.735502, 1.570796, 1.660984],accel_mss,speed_ms,0,blend_radius_m)
    movel([0.088826, -1.469540, -2.507271, -0.735578, 1.570796, 1.659622],accel_mss,speed_ms,0,blend_radius_m)
    movel([0.087603, -1.468975, -2.507744, -0.735670, 1.570796, 1.658399],accel_mss,speed_ms,0,blend_radius_m)
    movel([0.086506, -1.468282, -2.508324, -0.735783, 1.570796, 1.657302],accel_mss,speed_ms,0,blend_radius_m)
    movel([0.085524, -1.467429, -2.509037, -0.735923, 1.570796, 1.656320],accel_mss,speed_ms,0,blend_radius_m)
    movel([0.084643, -1.466383, -2.509910, -0.736096, 1.570796, 1.655440],accel_mss,speed_ms,0,blend_radius_m)
    movel([0.083856, -1.465107, -2.510972, -0.736310, 1.570796, 1.654652],accel_mss,speed_ms,0,blend_radius_m)
    movel([0.082558, -1.462229, -2.513360, -0.736801, 1.570796, 1.653354],accel_mss,speed_ms,0,blend_radius_m)
    movel([0.081589, -1.459156, -2.515894, -0.737340, 1.570796, 1.652385],accel_mss,speed_ms,0,blend_radius_m)
    movel([0.080918, -1.455920, -2.518546, -0.737923, 1.570796, 1.651715],accel_mss,speed_ms,0,blend_radius_m)
    movel([0.080512, -1.452560, -2.521284, -0.738545, 1.570796, 1.651308],accel_mss,speed_ms,0,blend_radius_m)
    movel([0.080370, -1.449728, -2.523578, -0.739083, 1.570796, 1.651166],accel_mss,speed_ms,0,blend_radius_m)
    movel([0.080382, -1.446835, -2.525908, -0.739646, 1.570796, 1.651178],accel_mss,speed_ms,0,blend_radius_m)
    movel([0.080742, -1.440899, -2.530650, -0.740841, 1.570796, 1.651538],accel_mss,speed_ms,0,blend_radius_m)
    movel([0.082666, -1.420006, -2.546911, -0.745472, 1.570796, 1.653463],accel_mss,speed_ms,0,blend_radius_m)
    movel([0.083026, -1.415559, -2.550287, -0.746543, 1.570796, 1.653822],accel_mss,speed_ms,0,blend_radius_m)
    movel([0.083283, -1.411110, -2.553636, -0.747644, 1.570796, 1.654079],accel_mss,speed_ms,0,blend_radius_m)
    movel([0.083368, -1.406699, -2.556926, -0.748764, 1.570796, 1.654164],accel_mss,speed_ms,0,blend_radius_m)
    movel([0.083208, -1.402363, -2.560132, -0.749894, 1.570796, 1.654004],accel_mss,speed_ms,0,blend_radius_m)
    movel([0.082733, -1.398144, -2.563225, -0.751019, 1.570796, 1.653529],accel_mss,speed_ms,0,blend_radius_m)
    movel([0.081869, -1.394085, -2.566177, -0.752127, 1.570796, 1.652665],accel_mss,speed_ms,0,blend_radius_m)
    movel([0.080970, -1.391249, -2.568224, -0.752916, 1.570796, 1.651766],accel_mss,speed_ms,0,blend_radius_m)
    movel([0.079818, -1.388453, -2.570232, -0.753704, 1.570796, 1.650614],accel_mss,speed_ms,0,blend_radius_m)
    movel([0.078401, -1.385756, -2.572157, -0.754476, 1.570796, 1.649197],accel_mss,speed_ms,0,blend_radius_m)
    movel([0.076708, -1.383220, -2.573958, -0.755211, 1.570796, 1.647504],accel_mss,speed_ms,0,blend_radius_m)
    movel([0.074731, -1.380903, -2.575595, -0.755891, 1.570796, 1.645528],accel_mss,speed_ms,0,blend_radius_m)
    movel([0.072462, -1.378866, -2.577029, -0.756495, 1.570796, 1.643258],accel_mss,speed_ms,0,blend_radius_m)
    movel([0.069890, -1.377173, -2.578215, -0.757001, 1.570796, 1.640686],accel_mss,speed_ms,0,blend_radius_m)
    movel([0.067014, -1.375884, -2.579115, -0.757390, 1.570796, 1.637810],accel_mss,speed_ms,0,blend_radius_m)
    movel([0.065543, -1.375455, -2.579415, -0.757520, 1.570796, 1.636339],accel_mss,speed_ms,0,blend_radius_m)
    movel([0.063973, -1.375163, -2.579618, -0.757608, 1.570796, 1.634770],accel_mss,speed_ms,0,blend_radius_m)
    movel([0.062316, -1.375024, -2.579715, -0.757650, 1.570796, 1.633112],accel_mss,speed_ms,0,blend_radius_m)
    movel([0.060588, -1.375048, -2.579698, -0.757643, 1.570796, 1.631385],accel_mss,speed_ms,0,blend_radius_m)
    movel([0.058808, -1.375244, -2.579562, -0.757584, 1.570796, 1.629604],accel_mss,speed_ms,0,blend_radius_m)
    movel([0.056985, -1.375626, -2.579295, -0.757468, 1.570796, 1.627782],accel_mss,speed_ms,0,blend_radius_m)
    movel([0.055140, -1.376201, -2.578894, -0.757294, 1.570796, 1.625936],accel_mss,speed_ms,0,blend_radius_m)
    movel([0.053288, -1.376983, -2.578348, -0.757058, 1.570796, 1.624085],accel_mss,speed_ms,0,blend_radius_m)
    speed_ms = 0.005
    movel([0.053288, -1.368176, -2.574340, -0.769873, 1.570796, 1.624085],accel_mss,speed_ms,0,blend_radius_m)
    speed_ms = 0.040
    movel([0.046440, -1.360211, -2.579790, -0.772387, 1.570796, 1.617236],accel_mss,speed_ms,0,blend_radius_m)
    speed_ms = 0.005
    movel([0.046440, -1.369074, -2.583834, -0.759481, 1.570796, 1.617236],accel_mss,speed_ms,0,blend_radius_m)
    speed_ms = 0.025
    movel([0.046162, -1.368001, -2.584571, -0.759817, 1.570796, 1.616958],accel_mss,speed_ms,0,blend_radius_m)
    movel([0.046032, -1.366863, -2.585351, -0.760175, 1.570796, 1.616829],accel_mss,speed_ms,0,blend_radius_m)
    movel([0.046134, -1.364445, -2.587003, -0.760941, 1.570796, 1.616930],accel_mss,speed_ms,0,blend_radius_m)
    movel([0.046579, -1.361899, -2.588733, -0.761756, 1.570796, 1.617375],accel_mss,speed_ms,0,blend_radius_m)
    movel([0.047196, -1.359315, -2.590481, -0.762594, 1.570796, 1.617993],accel_mss,speed_ms,0,blend_radius_m)
    speed_ms = 0.005
    movel([0.047196, -1.350384, -2.586394, -0.775610, 1.570796, 1.617993],accel_mss,speed_ms,0,blend_radius_m)
    speed_ms = 0.040
    movel([0.051241, -1.350725, -2.586167, -0.775496, 1.570796, 1.622038],accel_mss,speed_ms,0,blend_radius_m)
    speed_ms = 0.005
    movel([0.051241, -1.359653, -2.590252, -0.762483, 1.570796, 1.622038],accel_mss,speed_ms,0,blend_radius_m)
    speed_ms = 0.025
    movel([0.050674, -1.358844, -2.590798, -0.762747, 1.570796, 1.621470],accel_mss,speed_ms,0,blend_radius_m)
    movel([0.050253, -1.357967, -2.591388, -0.763034, 1.570796, 1.621050],accel_mss,speed_ms,0,blend_radius_m)
    movel([0.049813, -1.356029, -2.592688, -0.763672, 1.570796, 1.620609],accel_mss,speed_ms,0,blend_radius_m)
    movel([0.049852, -1.353892, -2.594116, -0.764381, 1.570796, 1.620648],accel_mss,speed_ms,0,blend_radius_m)
    movel([0.050298, -1.351602, -2.595639, -0.765148, 1.570796, 1.621095],accel_mss,speed_ms,0,blend_radius_m)
    movel([0.051081, -1.349210, -2.597222, -0.765958, 1.570796, 1.621878],accel_mss,speed_ms,0,blend_radius_m)
    movel([0.052129, -1.346769, -2.598828, -0.766791, 1.570796, 1.622925],accel_mss,speed_ms,0,blend_radius_m)
    movel([0.053366, -1.344331, -2.600426, -0.767633, 1.570796, 1.624162],accel_mss,speed_ms,0,blend_radius_m)
    movel([0.054720, -1.341950, -2.601977, -0.768462, 1.570796, 1.625516],accel_mss,speed_ms,0,blend_radius_m)
    speed_ms = 0.005
    movel([0.054720, -1.332903, -2.597814, -0.781673, 1.570796, 1.625516],accel_mss,speed_ms,0,blend_radius_m)
    speed_ms = 0.040
    movel([0.072655, -1.312994, -2.610316, -0.789079, 1.570796, 1.643451],accel_mss,speed_ms,0,blend_radius_m)
    speed_ms = 0.005
    movel([0.072655, -1.322169, -2.614569, -0.775652, 1.570796, 1.643451],accel_mss,speed_ms,0,blend_radius_m)
    speed_ms = 0.025
    movel([0.070826, -1.323587, -2.613684, -0.775118, 1.570796, 1.641623],accel_mss,speed_ms,0,blend_radius_m)
    movel([0.069012, -1.325143, -2.612709, -0.774537, 1.570796, 1.639808],accel_mss,speed_ms,0,blend_radius_m)
    movel([0.067241, -1.326813, -2.611660, -0.773916, 1.570796, 1.638037],accel_mss,speed_ms,0,blend_radius_m)
    movel([0.065533, -1.328576, -2.610548, -0.773265, 1.570796, 1.636329],accel_mss,speed_ms,0,blend_radius_m)
    movel([0.063919, -1.330414, -2.609385, -0.772590, 1.570796, 1.634715],accel_mss,speed_ms,0,blend_radius_m)
    movel([0.062422, -1.332301, -2.608185, -0.771902, 1.570796, 1.633218],accel_mss,speed_ms,0,blend_radius_m)
    movel([0.061068, -1.334221, -2.606960, -0.771208, 1.570796, 1.631864],accel_mss,speed_ms,0,blend_radius_m)
    movel([0.059882, -1.336154, -2.605721, -0.770513, 1.570796, 1.630678],accel_mss,speed_ms,0,blend_radius_m)
    movel([0.058887, -1.338076, -2.604485, -0.769828, 1.570796, 1.629684],accel_mss,speed_ms,0,blend_radius_m)
    movel([0.058108, -1.339972, -2.603260, -0.769157, 1.570796, 1.628904],accel_mss,speed_ms,0,blend_radius_m)
    movel([0.057567, -1.341820, -2.602062, -0.768508, 1.570796, 1.628364],accel_mss,speed_ms,0,blend_radius_m)
    movel([0.057288, -1.343602, -2.600902, -0.767886, 1.570796, 1.628084],accel_mss,speed_ms,0,blend_radius_m)
    movel([0.057295, -1.345298, -2.599793, -0.767298, 1.570796, 1.628091],accel_mss,speed_ms,0,blend_radius_m)
    movel([0.057612, -1.346892, -2.598748, -0.766749, 1.570796, 1.628408],accel_mss,speed_ms,0,blend_radius_m)
    movel([0.058258, -1.348366, -2.597778, -0.766245, 1.570796, 1.629054],accel_mss,speed_ms,0,blend_radius_m)
    movel([0.059259, -1.349702, -2.596896, -0.765790, 1.570796, 1.630055],accel_mss,speed_ms,0,blend_radius_m)
    speed_ms = 0.005
    movel([0.059259, -1.340707, -2.592767, -0.778915, 1.570796, 1.630055],accel_mss,speed_ms,0,blend_radius_m)
    speed_ms = 0.040
    movel([0.068039, -1.334366, -2.596873, -0.781149, 1.570796, 1.638836],accel_mss,speed_ms,0,blend_radius_m)
    speed_ms = 0.005
    movel([0.068039, -1.343403, -2.601031, -0.767955, 1.570796, 1.638836],accel_mss,speed_ms,0,blend_radius_m)
    speed_ms = 0.025
    movel([0.067695, -1.342130, -2.601860, -0.768399, 1.570796, 1.638492],accel_mss,speed_ms,0,blend_radius_m)
    movel([0.067496, -1.340778, -2.602738, -0.768873, 1.570796, 1.638292],accel_mss,speed_ms,0,blend_radius_m)
    movel([0.067439, -1.339363, -2.603654, -0.769372, 1.570796, 1.638235],accel_mss,speed_ms,0,blend_radius_m)
    movel([0.067526, -1.337893, -2.604603, -0.769893, 1.570796, 1.638322],accel_mss,speed_ms,0,blend_radius_m)
    movel([0.067753, -1.336383, -2.605575, -0.770431, 1.570796, 1.638550],accel_mss,speed_ms,0,blend_radius_m)
    movel([0.068124, -1.334842, -2.606563, -0.770984, 1.570796, 1.638920],accel_mss,speed_ms,0,blend_radius_m)
    movel([0.068637, -1.333279, -2.607562, -0.771548, 1.570796, 1.639433],accel_mss,speed_ms,0,blend_radius_m)
    movel([0.069290, -1.331712, -2.608561, -0.772117, 1.570796, 1.640086],accel_mss,speed_ms,0,blend_radius_m)
    movel([0.070082, -1.330148, -2.609553, -0.772687, 1.570796, 1.640879],accel_mss,speed_ms,0,blend_radius_m)
    movel([0.071017, -1.328600, -2.610533, -0.773256, 1.570796, 1.641813],accel_mss,speed_ms,0,blend_radius_m)
    movel([0.072087, -1.327085, -2.611489, -0.773815, 1.570796, 1.642883],accel_mss,speed_ms,0,blend_radius_m)
    movel([0.073298, -1.325609, -2.612417, -0.774363, 1.570796, 1.644094],accel_mss,speed_ms,0,blend_radius_m)
    movel([0.074647, -1.324187, -2.613308, -0.774894, 1.570796, 1.645443],accel_mss,speed_ms,0,blend_radius_m)
    movel([0.076132, -1.322833, -2.614155, -0.775402, 1.570796, 1.646928],accel_mss,speed_ms,0,blend_radius_m)
    movel([0.077752, -1.321560, -2.614948, -0.775881, 1.570796, 1.648548],accel_mss,speed_ms,0,blend_radius_m)
    movel([0.079504, -1.320381, -2.615681, -0.776327, 1.570796, 1.650300],accel_mss,speed_ms,0,blend_radius_m)
    movel([0.081276, -1.319378, -2.616302, -0.776708, 1.570796, 1.652073],accel_mss,speed_ms,0,blend_radius_m)
    movel([0.083056, -1.318553, -2.616813, -0.777023, 1.570796, 1.653852],accel_mss,speed_ms,0,blend_radius_m)
    movel([0.084829, -1.317900, -2.617217, -0.777272, 1.570796, 1.655625],accel_mss,speed_ms,0,blend_radius_m)
    movel([0.086589, -1.317413, -2.617518, -0.777459, 1.570796, 1.657386],accel_mss,speed_ms,0,blend_radius_m)
    movel([0.088324, -1.317086, -2.617719, -0.777584, 1.570796, 1.659120],accel_mss,speed_ms,0,blend_radius_m)
    movel([0.090019, -1.316916, -2.617823, -0.777649, 1.570796, 1.660815],accel_mss,speed_ms,0,blend_radius_m)
    movel([0.091669, -1.316893, -2.617838, -0.777658, 1.570796, 1.662465],accel_mss,speed_ms,0,blend_radius_m)
    movel([0.093255, -1.317014, -2.617763, -0.777612, 1.570796, 1.664052],accel_mss,speed_ms,0,blend_radius_m)
    movel([0.094774, -1.317271, -2.617605, -0.777513, 1.570796, 1.665570],accel_mss,speed_ms,0,blend_radius_m)
    movel([0.097561, -1.318165, -2.617053, -0.777171, 1.570796, 1.668358],accel_mss,speed_ms,0,blend_radius_m)
    movel([0.098805, -1.318790, -2.616666, -0.776932, 1.570796, 1.669601],accel_mss,speed_ms,0,blend_radius_m)
    movel([0.100955, -1.320357, -2.615696, -0.776336, 1.570796, 1.671751],accel_mss,speed_ms,0,blend_radius_m)
    movel([0.101839, -1.321283, -2.615120, -0.775986, 1.570796, 1.672635],accel_mss,speed_ms,0,blend_radius_m)
    movel([0.102581, -1.322297, -2.614489, -0.775603, 1.570796, 1.673377],accel_mss,speed_ms,0,blend_radius_m)
    speed_ms = 0.005
    movel([0.102581, -1.313124, -2.610237, -0.789029, 1.570796, 1.673377],accel_mss,speed_ms,0,blend_radius_m)
    speed_ms = 0.040
    movel([0.110269, -1.321109, -2.605284, -0.785997, 1.570796, 1.681065],accel_mss,speed_ms,0,blend_radius_m)
    speed_ms = 0.005
    movel([0.110269, -1.330232, -2.609500, -0.772657, 1.570796, 1.681065],accel_mss,speed_ms,0,blend_radius_m)
    speed_ms = 0.025
    movel([0.109196, -1.328664, -2.610493, -0.773232, 1.570796, 1.679992],accel_mss,speed_ms,0,blend_radius_m)
    movel([0.107816, -1.327375, -2.611306, -0.773708, 1.570796, 1.678612],accel_mss,speed_ms,0,blend_radius_m)
    movel([0.106160, -1.326376, -2.611935, -0.774078, 1.570796, 1.676957],accel_mss,speed_ms,0,blend_radius_m)
    movel([0.104255, -1.325678, -2.612373, -0.774337, 1.570796, 1.675051],accel_mss,speed_ms,0,blend_radius_m)
    movel([0.102138, -1.325289, -2.612618, -0.774482, 1.570796, 1.672934],accel_mss,speed_ms,0,blend_radius_m)
    movel([0.099836, -1.325221, -2.612661, -0.774508, 1.570796, 1.670633],accel_mss,speed_ms,0,blend_radius_m)
    movel([0.097387, -1.325480, -2.612498, -0.774411, 1.570796, 1.668183],accel_mss,speed_ms,0,blend_radius_m)
    movel([0.094817, -1.326075, -2.612124, -0.774190, 1.570796, 1.665613],accel_mss,speed_ms,0,blend_radius_m)
    movel([0.092168, -1.327011, -2.611535, -0.773843, 1.570796, 1.662964],accel_mss,speed_ms,0,blend_radius_m)
    movel([0.089499, -1.328276, -2.610738, -0.773375, 1.570796, 1.660295],accel_mss,speed_ms,0,blend_radius_m)
    movel([0.086911, -1.329833, -2.609753, -0.772803, 1.570796, 1.657708],accel_mss,speed_ms,0,blend_radius_m)
    movel([0.084515, -1.331644, -2.608603, -0.772141, 1.570796, 1.655311],accel_mss,speed_ms,0,blend_radius_m)
    movel([0.082407, -1.333677, -2.607308, -0.771404, 1.570796, 1.653204],accel_mss,speed_ms,0,blend_radius_m)
    movel([0.081497, -1.334764, -2.606613, -0.771012, 1.570796, 1.652293],accel_mss,speed_ms,0,blend_radius_m)
    movel([0.080695, -1.335891, -2.605891, -0.770608, 1.570796, 1.651491],accel_mss,speed_ms,0,blend_radius_m)
    movel([0.080015, -1.337055, -2.605142, -0.770191, 1.570796, 1.650811],accel_mss,speed_ms,0,blend_radius_m)
    movel([0.079472, -1.338255, -2.604370, -0.769765, 1.570796, 1.650269],accel_mss,speed_ms,0,blend_radius_m)
    movel([0.079075, -1.339481, -2.603578, -0.769330, 1.570796, 1.649871],accel_mss,speed_ms,0,blend_radius_m)
    movel([0.078840, -1.340729, -2.602770, -0.768890, 1.570796, 1.649636],accel_mss,speed_ms,0,blend_radius_m)
    speed_ms = 0.005
    movel([0.078840, -1.331674, -2.598601, -0.782115, 1.570796, 1.649636],accel_mss,speed_ms,0,blend_radius_m)
    speed_ms = 0.040
    movel([0.093268, -1.333460, -2.597456, -0.781473, 1.570796, 1.664064],accel_mss,speed_ms,0,blend_radius_m)
    speed_ms = 0.005
    movel([0.093268, -1.342503, -2.601617, -0.768269, 1.570796, 1.664064],accel_mss,speed_ms,0,blend_radius_m)
    speed_ms = 0.025
    movel([0.095033, -1.341187, -2.602473, -0.768729, 1.570796, 1.665829],accel_mss,speed_ms,0,blend_radius_m)
    movel([0.096890, -1.340087, -2.603186, -0.769116, 1.570796, 1.667686],accel_mss,speed_ms,0,blend_radius_m)
    movel([0.098808, -1.339199, -2.603760, -0.769430, 1.570796, 1.669605],accel_mss,speed_ms,0,blend_radius_m)
    movel([0.100748, -1.338523, -2.604197, -0.769669, 1.570796, 1.671544],accel_mss,speed_ms,0,blend_radius_m)
    movel([0.102675, -1.338054, -2.604499, -0.769836, 1.570796, 1.673471],accel_mss,speed_ms,0,blend_radius_m)
    movel([0.104550, -1.337786, -2.604672, -0.769931, 1.570796, 1.675346],accel_mss,speed_ms,0,blend_radius_m)
    movel([0.106343, -1.337716, -2.604717, -0.769956, 1.570796, 1.677139],accel_mss,speed_ms,0,blend_radius_m)
    movel([0.108012, -1.337837, -2.604639, -0.769913, 1.570796, 1.678808],accel_mss,speed_ms,0,blend_radius_m)
    movel([0.109822, -1.338281, -2.604353, -0.769755, 1.570796, 1.680618],accel_mss,speed_ms,0,blend_radius_m)
    movel([0.111204, -1.339034, -2.603867, -0.769488, 1.570796, 1.682000],accel_mss,speed_ms,0,blend_radius_m)
    movel([0.112205, -1.340061, -2.603203, -0.769125, 1.570796, 1.683001],accel_mss,speed_ms,0,blend_radius_m)
    movel([0.112862, -1.341332, -2.602378, -0.768678, 1.570796, 1.683659],accel_mss,speed_ms,0,blend_radius_m)
    movel([0.113220, -1.342808, -2.601419, -0.768162, 1.570796, 1.684017],accel_mss,speed_ms,0,blend_radius_m)
    movel([0.113322, -1.344460, -2.600341, -0.767588, 1.570796, 1.684118],accel_mss,speed_ms,0,blend_radius_m)
    movel([0.113208, -1.346250, -2.599169, -0.766970, 1.570796, 1.684005],accel_mss,speed_ms,0,blend_radius_m)
    movel([0.112925, -1.348147, -2.597922, -0.766320, 1.570796, 1.683721],accel_mss,speed_ms,0,blend_radius_m)
    speed_ms = 0.005
    movel([0.112925, -1.339141, -2.593786, -0.779462, 1.570796, 1.683721],accel_mss,speed_ms,0,blend_radius_m)
    speed_ms = 0.040
    movel([0.099676, -1.341605, -2.592181, -0.778603, 1.570796, 1.670472],accel_mss,speed_ms,0,blend_radius_m)
    speed_ms = 0.005
    movel([0.099676, -1.350595, -2.596306, -0.765488, 1.570796, 1.670472],accel_mss,speed_ms,0,blend_radius_m)
    speed_ms = 0.025
    movel([0.101479, -1.350410, -2.596428, -0.765551, 1.570796, 1.672275],accel_mss,speed_ms,0,blend_radius_m)
    movel([0.103139, -1.350430, -2.596415, -0.765544, 1.570796, 1.673935],accel_mss,speed_ms,0,blend_radius_m)
    movel([0.104656, -1.350648, -2.596271, -0.765470, 1.570796, 1.675452],accel_mss,speed_ms,0,blend_radius_m)
    movel([0.106032, -1.351045, -2.596008, -0.765336, 1.570796, 1.676828],accel_mss,speed_ms,0,blend_radius_m)
    movel([0.107267, -1.351611, -2.595633, -0.765145, 1.570796, 1.678063],accel_mss,speed_ms,0,blend_radius_m)
    movel([0.108360, -1.352330, -2.595155, -0.764904, 1.570796, 1.679157],accel_mss,speed_ms,0,blend_radius_m)
    movel([0.109317, -1.353190, -2.594583, -0.764615, 1.570796, 1.680113],accel_mss,speed_ms,0,blend_radius_m)
    movel([0.110132, -1.354180, -2.593924, -0.764285, 1.570796, 1.680928],accel_mss,speed_ms,0,blend_radius_m)
    movel([0.110813, -1.355283, -2.593187, -0.763919, 1.570796, 1.681609],accel_mss,speed_ms,0,blend_radius_m)
    movel([0.111359, -1.356487, -2.592381, -0.763521, 1.570796, 1.682156],accel_mss,speed_ms,0,blend_radius_m)
    movel([0.111771, -1.357779, -2.591514, -0.763096, 1.570796, 1.682567],accel_mss,speed_ms,0,blend_radius_m)
    movel([0.112052, -1.359145, -2.590595, -0.762649, 1.570796, 1.682848],accel_mss,speed_ms,0,blend_radius_m)
    movel([0.112203, -1.360573, -2.589631, -0.762185, 1.570796, 1.682999],accel_mss,speed_ms,0,blend_radius_m)
    movel([0.112122, -1.363559, -2.587606, -0.761224, 1.570796, 1.682918],accel_mss,speed_ms,0,blend_radius_m)
    movel([0.111891, -1.365095, -2.586560, -0.760734, 1.570796, 1.682688],accel_mss,speed_ms,0,blend_radius_m)
    movel([0.111752, -1.364641, -2.586869, -0.760878, 1.570796, 1.682549],accel_mss,speed_ms,0,blend_radius_m)
    speed_ms = 0.005
    movel([0.111752, -1.355748, -2.582807, -0.773834, 1.570796, 1.682549],accel_mss,speed_ms,0,blend_radius_m)
    speed_ms = 0.040
    movel([0.123071, -1.359054, -2.580575, -0.772760, 1.570796, 1.693867],accel_mss,speed_ms,0,blend_radius_m)
    speed_ms = 0.005
    movel([0.123071, -1.367925, -2.584623, -0.759841, 1.570796, 1.693867],accel_mss,speed_ms,0,blend_radius_m)
    speed_ms = 0.025
    movel([0.121545, -1.370024, -2.583179, -0.759185, 1.570796, 1.692342],accel_mss,speed_ms,0,blend_radius_m)
    movel([0.120248, -1.372172, -2.581695, -0.758521, 1.570796, 1.691045],accel_mss,speed_ms,0,blend_radius_m)
    movel([0.119128, -1.374343, -2.580188, -0.757857, 1.570796, 1.689924],accel_mss,speed_ms,0,blend_radius_m)
    movel([0.118129, -1.376514, -2.578675, -0.757199, 1.570796, 1.688925],accel_mss,speed_ms,0,blend_radius_m)
    movel([0.117153, -1.378898, -2.577006, -0.756485, 1.570796, 1.687949],accel_mss,speed_ms,0,blend_radius_m)
    movel([0.116786, -1.380072, -2.576180, -0.756136, 1.570796, 1.687582],accel_mss,speed_ms,0,blend_radius_m)
    movel([0.116551, -1.381222, -2.575370, -0.755797, 1.570796, 1.687348],accel_mss,speed_ms,0,blend_radius_m)
    movel([0.116481, -1.382333, -2.574586, -0.755470, 1.570796, 1.687278],accel_mss,speed_ms,0,blend_radius_m)
    movel([0.116613, -1.383365, -2.573855, -0.755169, 1.570796, 1.687409],accel_mss,speed_ms,0,blend_radius_m)
    movel([0.116973, -1.384264, -2.573218, -0.754907, 1.570796, 1.687769],accel_mss,speed_ms,0,blend_radius_m)
    movel([0.117585, -1.384985, -2.572706, -0.754698, 1.570796, 1.688382],accel_mss,speed_ms,0,blend_radius_m)
    movel([0.118935, -1.385766, -2.572150, -0.754473, 1.570796, 1.689731],accel_mss,speed_ms,0,blend_radius_m)
    movel([0.119601, -1.386159, -2.571870, -0.754360, 1.570796, 1.690397],accel_mss,speed_ms,0,blend_radius_m)
    movel([0.120138, -1.386668, -2.571507, -0.754214, 1.570796, 1.690934],accel_mss,speed_ms,0,blend_radius_m)
    movel([0.120477, -1.387472, -2.570933, -0.753984, 1.570796, 1.691273],accel_mss,speed_ms,0,blend_radius_m)
    movel([0.120547, -1.388501, -2.570197, -0.753691, 1.570796, 1.691343],accel_mss,speed_ms,0,blend_radius_m)
    movel([0.120405, -1.389692, -2.569344, -0.753353, 1.570796, 1.691201],accel_mss,speed_ms,0,blend_radius_m)
    movel([0.120104, -1.390978, -2.568420, -0.752992, 1.570796, 1.690900],accel_mss,speed_ms,0,blend_radius_m)
    movel([0.119240, -1.393583, -2.566540, -0.752266, 1.570796, 1.690037],accel_mss,speed_ms,0,blend_radius_m)
    movel([0.116329, -1.400820, -2.561267, -0.750302, 1.570796, 1.687125],accel_mss,speed_ms,0,blend_radius_m)
    movel([0.114314, -1.405791, -2.557600, -0.748998, 1.570796, 1.685111],accel_mss,speed_ms,0,blend_radius_m)
    movel([0.113817, -1.407309, -2.556472, -0.748607, 1.570796, 1.684613],accel_mss,speed_ms,0,blend_radius_m)
    movel([0.113407, -1.408921, -2.555272, -0.748196, 1.570796, 1.684203],accel_mss,speed_ms,0,blend_radius_m)
    movel([0.112896, -1.412284, -2.552755, -0.747350, 1.570796, 1.683692],accel_mss,speed_ms,0,blend_radius_m)
    movel([0.112821, -1.413966, -2.551490, -0.746933, 1.570796, 1.683617],accel_mss,speed_ms,0,blend_radius_m)
    movel([0.112885, -1.415600, -2.550256, -0.746533, 1.570796, 1.683682],accel_mss,speed_ms,0,blend_radius_m)
    movel([0.113098, -1.417154, -2.549080, -0.746155, 1.570796, 1.683895],accel_mss,speed_ms,0,blend_radius_m)
    movel([0.113474, -1.418593, -2.547987, -0.745809, 1.570796, 1.684270],accel_mss,speed_ms,0,blend_radius_m)
    movel([0.114025, -1.419881, -2.547006, -0.745502, 1.570796, 1.684821],accel_mss,speed_ms,0,blend_radius_m)
    movel([0.114762, -1.420989, -2.546160, -0.745239, 1.570796, 1.685558],accel_mss,speed_ms,0,blend_radius_m)
    movel([0.115701, -1.421880, -2.545480, -0.745030, 1.570796, 1.686498],accel_mss,speed_ms,0,blend_radius_m)
    movel([0.116854, -1.422521, -2.544988, -0.744879, 1.570796, 1.687651],accel_mss,speed_ms,0,blend_radius_m)
    movel([0.118233, -1.422880, -2.544713, -0.744796, 1.570796, 1.689029],accel_mss,speed_ms,0,blend_radius_m)
    movel([0.119854, -1.422922, -2.544681, -0.744786, 1.570796, 1.690650],accel_mss,speed_ms,0,blend_radius_m)
    movel([0.121731, -1.422614, -2.544917, -0.744858, 1.570796, 1.692527],accel_mss,speed_ms,0,blend_radius_m)
    movel([0.123879, -1.421921, -2.545448, -0.745020, 1.570796, 1.694676],accel_mss,speed_ms,0,blend_radius_m)
    movel([0.125555, -1.421175, -2.546019, -0.745195, 1.570796, 1.696351],accel_mss,speed_ms,0,blend_radius_m)
    movel([0.127184, -1.420287, -2.546697, -0.745405, 1.570796, 1.697980],accel_mss,speed_ms,0,blend_radius_m)
    movel([0.128776, -1.419279, -2.547465, -0.745645, 1.570796, 1.699572],accel_mss,speed_ms,0,blend_radius_m)
    movel([0.130334, -1.418175, -2.548305, -0.745909, 1.570796, 1.701131],accel_mss,speed_ms,0,blend_radius_m)
    movel([0.133374, -1.415778, -2.550122, -0.746489, 1.570796, 1.704171],accel_mss,speed_ms,0,blend_radius_m)
    movel([0.136352, -1.413287, -2.552001, -0.747101, 1.570796, 1.707148],accel_mss,speed_ms,0,blend_radius_m)
    movel([0.139412, -1.410842, -2.553836, -0.747711, 1.570796, 1.710209],accel_mss,speed_ms,0,blend_radius_m)
    movel([0.141009, -1.409685, -2.554702, -0.748002, 1.570796, 1.711805],accel_mss,speed_ms,0,blend_radius_m)
    movel([0.142640, -1.408615, -2.555500, -0.748274, 1.570796, 1.713437],accel_mss,speed_ms,0,blend_radius_m)
    movel([0.144300, -1.407659, -2.556212, -0.748518, 1.570796, 1.715097],accel_mss,speed_ms,0,blend_radius_m)
    movel([0.145983, -1.406851, -2.556813, -0.748725, 1.570796, 1.716779],accel_mss,speed_ms,0,blend_radius_m)
    movel([0.147676, -1.406221, -2.557281, -0.748887, 1.570796, 1.718473],accel_mss,speed_ms,0,blend_radius_m)
    movel([0.149377, -1.405801, -2.557592, -0.748996, 1.570796, 1.720174],accel_mss,speed_ms,0,blend_radius_m)
    movel([0.152990, -1.405406, -2.557885, -0.749098, 1.570796, 1.723787],accel_mss,speed_ms,0,blend_radius_m)
    movel([0.154212, -1.405191, -2.558044, -0.749154, 1.570796, 1.725008],accel_mss,speed_ms,0,blend_radius_m)
    movel([0.155484, -1.404787, -2.558343, -0.749259, 1.570796, 1.726281],accel_mss,speed_ms,0,blend_radius_m)
    movel([0.156737, -1.404161, -2.558806, -0.749422, 1.570796, 1.727533],accel_mss,speed_ms,0,blend_radius_m)
    movel([0.157844, -1.403331, -2.559419, -0.749639, 1.570796, 1.728640],accel_mss,speed_ms,0,blend_radius_m)
    movel([0.158305, -1.402841, -2.559780, -0.749768, 1.570796, 1.729101],accel_mss,speed_ms,0,blend_radius_m)
    movel([0.158684, -1.402306, -2.560174, -0.749909, 1.570796, 1.729481],accel_mss,speed_ms,0,blend_radius_m)
    speed_ms = 0.005
    movel([0.158684, -1.393683, -2.556277, -0.762429, 1.570796, 1.729481],accel_mss,speed_ms,0,blend_radius_m)
    speed_ms = 0.040
    movel([0.163841, -1.383356, -2.563702, -0.765331, 1.570796, 1.734638],accel_mss,speed_ms,0,blend_radius_m)
    speed_ms = 0.005
    movel([0.163841, -1.392055, -2.567644, -0.752690, 1.570796, 1.734638],accel_mss,speed_ms,0,blend_radius_m)
    speed_ms = 0.025
    movel([0.164253, -1.392182, -2.567552, -0.752655, 1.570796, 1.735050],accel_mss,speed_ms,0,blend_radius_m)
    movel([0.164327, -1.392616, -2.567239, -0.752534, 1.570796, 1.735124],accel_mss,speed_ms,0,blend_radius_m)
    movel([0.164108, -1.393172, -2.566837, -0.752380, 1.570796, 1.734904],accel_mss,speed_ms,0,blend_radius_m)
    movel([0.163650, -1.393670, -2.566477, -0.752242, 1.570796, 1.734446],accel_mss,speed_ms,0,blend_radius_m)
    movel([0.163068, -1.394005, -2.566235, -0.752149, 1.570796, 1.733864],accel_mss,speed_ms,0,blend_radius_m)
    movel([0.162458, -1.394227, -2.566074, -0.752088, 1.570796, 1.733254],accel_mss,speed_ms,0,blend_radius_m)
    movel([0.161217, -1.394556, -2.565835, -0.751997, 1.570796, 1.732013],accel_mss,speed_ms,0,blend_radius_m)
    movel([0.160327, -1.394883, -2.565598, -0.751907, 1.570796, 1.731124],accel_mss,speed_ms,0,blend_radius_m)
    movel([0.159463, -1.395317, -2.565284, -0.751789, 1.570796, 1.730260],accel_mss,speed_ms,0,blend_radius_m)
    movel([0.157805, -1.396432, -2.564474, -0.751484, 1.570796, 1.728601],accel_mss,speed_ms,0,blend_radius_m)
    movel([0.156242, -1.397767, -2.563501, -0.751121, 1.570796, 1.727038],accel_mss,speed_ms,0,blend_radius_m)
    movel([0.154774, -1.399178, -2.562470, -0.750741, 1.570796, 1.725570],accel_mss,speed_ms,0,blend_radius_m)
    movel([0.154445, -1.399538, -2.562206, -0.750645, 1.570796, 1.725242],accel_mss,speed_ms,0,blend_radius_m)
    movel([0.154265, -1.399912, -2.561932, -0.750544, 1.570796, 1.725061],accel_mss,speed_ms,0,blend_radius_m)
    movel([0.154397, -1.400249, -2.561686, -0.750455, 1.570796, 1.725193],accel_mss,speed_ms,0,blend_radius_m)
    movel([0.154768, -1.400424, -2.561557, -0.750408, 1.570796, 1.725564],accel_mss,speed_ms,0,blend_radius_m)
    movel([0.155724, -1.400624, -2.561410, -0.750354, 1.570796, 1.726520],accel_mss,speed_ms,0,blend_radius_m)
    movel([0.156759, -1.400676, -2.561372, -0.750341, 1.570796, 1.727556],accel_mss,speed_ms,0,blend_radius_m)
    movel([0.157857, -1.400588, -2.561437, -0.750364, 1.570796, 1.728653],accel_mss,speed_ms,0,blend_radius_m)
    movel([0.158997, -1.400359, -2.561605, -0.750425, 1.570796, 1.729793],accel_mss,speed_ms,0,blend_radius_m)
    movel([0.160153, -1.400003, -2.561866, -0.750520, 1.570796, 1.730949],accel_mss,speed_ms,0,blend_radius_m)
    movel([0.161308, -1.399517, -2.562221, -0.750650, 1.570796, 1.732104],accel_mss,speed_ms,0,blend_radius_m)
    movel([0.162437, -1.398913, -2.562664, -0.750812, 1.570796, 1.733233],accel_mss,speed_ms,0,blend_radius_m)
    movel([0.163521, -1.398190, -2.563192, -0.751007, 1.570796, 1.734317],accel_mss,speed_ms,0,blend_radius_m)
    movel([0.163400, -1.398772, -2.562767, -0.750850, 1.570796, 1.734197],accel_mss,speed_ms,0,blend_radius_m)
    movel([0.163574, -1.399245, -2.562421, -0.750723, 1.570796, 1.734370],accel_mss,speed_ms,0,blend_radius_m)
    movel([0.163975, -1.399570, -2.562183, -0.750636, 1.570796, 1.734772],accel_mss,speed_ms,0,blend_radius_m)
    movel([0.164536, -1.399706, -2.562084, -0.750600, 1.570796, 1.735332],accel_mss,speed_ms,0,blend_radius_m)
    movel([0.165181, -1.399652, -2.562123, -0.750614, 1.570796, 1.735977],accel_mss,speed_ms,0,blend_radius_m)
    movel([0.165864, -1.399463, -2.562261, -0.750665, 1.570796, 1.736660],accel_mss,speed_ms,0,blend_radius_m)
    movel([0.167238, -1.398820, -2.562732, -0.750837, 1.570796, 1.738034],accel_mss,speed_ms,0,blend_radius_m)
    movel([0.168922, -1.397751, -2.563512, -0.751126, 1.570796, 1.739718],accel_mss,speed_ms,0,blend_radius_m)
    movel([0.170487, -1.396493, -2.564429, -0.751467, 1.570796, 1.741283],accel_mss,speed_ms,0,blend_radius_m)
    movel([0.171890, -1.395085, -2.565452, -0.751852, 1.570796, 1.742686],accel_mss,speed_ms,0,blend_radius_m)
    movel([0.173086, -1.393566, -2.566552, -0.752271, 1.570796, 1.743883],accel_mss,speed_ms,0,blend_radius_m)
    movel([0.173408, -1.393031, -2.566939, -0.752419, 1.570796, 1.744204],accel_mss,speed_ms,0,blend_radius_m)
    movel([0.173512, -1.392525, -2.567304, -0.752559, 1.570796, 1.744308],accel_mss,speed_ms,0,blend_radius_m)
    movel([0.173342, -1.392209, -2.567532, -0.752647, 1.570796, 1.744138],accel_mss,speed_ms,0,blend_radius_m)
    movel([0.173026, -1.392001, -2.567682, -0.752705, 1.570796, 1.743822],accel_mss,speed_ms,0,blend_radius_m)
    movel([0.171784, -1.391522, -2.568028, -0.752839, 1.570796, 1.742580],accel_mss,speed_ms,0,blend_radius_m)
    movel([0.169317, -1.390857, -2.568506, -0.753025, 1.570796, 1.740113],accel_mss,speed_ms,0,blend_radius_m)
    movel([0.168208, -1.390213, -2.568969, -0.753206, 1.570796, 1.739004],accel_mss,speed_ms,0,blend_radius_m)
    movel([0.169987, -1.388647, -2.570093, -0.753649, 1.570796, 1.740783],accel_mss,speed_ms,0,blend_radius_m)
    movel([0.170968, -1.387993, -2.570561, -0.753835, 1.570796, 1.741765],accel_mss,speed_ms,0,blend_radius_m)
    movel([0.171997, -1.387480, -2.570928, -0.753981, 1.570796, 1.742793],accel_mss,speed_ms,0,blend_radius_m)
    movel([0.172714, -1.387243, -2.571097, -0.754049, 1.570796, 1.743511],accel_mss,speed_ms,0,blend_radius_m)
    movel([0.173467, -1.387093, -2.571204, -0.754092, 1.570796, 1.744263],accel_mss,speed_ms,0,blend_radius_m)
    movel([0.174827, -1.387075, -2.571216, -0.754097, 1.570796, 1.745623],accel_mss,speed_ms,0,blend_radius_m)
    movel([0.175552, -1.387393, -2.570990, -0.754006, 1.570796, 1.746349],accel_mss,speed_ms,0,blend_radius_m)
    movel([0.175768, -1.387685, -2.570781, -0.753923, 1.570796, 1.746564],accel_mss,speed_ms,0,blend_radius_m)
    movel([0.175839, -1.388063, -2.570511, -0.753815, 1.570796, 1.746635],accel_mss,speed_ms,0,blend_radius_m)
    movel([0.175694, -1.388624, -2.570109, -0.753656, 1.570796, 1.746490],accel_mss,speed_ms,0,blend_radius_m)
    movel([0.175338, -1.389191, -2.569703, -0.753495, 1.570796, 1.746134],accel_mss,speed_ms,0,blend_radius_m)
    movel([0.174287, -1.390246, -2.568946, -0.753197, 1.570796, 1.745084],accel_mss,speed_ms,0,blend_radius_m)
    speed_ms = 0.005
    movel([0.174287, -1.381535, -2.564996, -0.765859, 1.570796, 1.745084],accel_mss,speed_ms,0,blend_radius_m)
    speed_ms = 0.040
    movel([0.180508, -1.341126, -2.592494, -0.778769, 1.570796, 1.751304],accel_mss,speed_ms,0,blend_radius_m)
    speed_ms = 0.005
    movel([0.180508, -1.350119, -2.596621, -0.765649, 1.570796, 1.751304],accel_mss,speed_ms,0,blend_radius_m)
    speed_ms = 0.025
    movel([0.181283, -1.349654, -2.596929, -0.765807, 1.570796, 1.752080],accel_mss,speed_ms,0,blend_radius_m)
    movel([0.182076, -1.349311, -2.597155, -0.765923, 1.570796, 1.752872],accel_mss,speed_ms,0,blend_radius_m)
    movel([0.182867, -1.349087, -2.597302, -0.765999, 1.570796, 1.753663],accel_mss,speed_ms,0,blend_radius_m)
    movel([0.184384, -1.348980, -2.597373, -0.766036, 1.570796, 1.755181],accel_mss,speed_ms,0,blend_radius_m)
    movel([0.185075, -1.349087, -2.597303, -0.765999, 1.570796, 1.755872],accel_mss,speed_ms,0,blend_radius_m)
    movel([0.186237, -1.349601, -2.596964, -0.765825, 1.570796, 1.757033],accel_mss,speed_ms,0,blend_radius_m)
    movel([0.187058, -1.350442, -2.596408, -0.765540, 1.570796, 1.757854],accel_mss,speed_ms,0,blend_radius_m)
    movel([0.187587, -1.351509, -2.595700, -0.765180, 1.570796, 1.758383],accel_mss,speed_ms,0,blend_radius_m)
    movel([0.187873, -1.352735, -2.594886, -0.764768, 1.570796, 1.758670],accel_mss,speed_ms,0,blend_radius_m)
    movel([0.187965, -1.354052, -2.594009, -0.764328, 1.570796, 1.758762],accel_mss,speed_ms,0,blend_radius_m)
    movel([0.187829, -1.356140, -2.592614, -0.763635, 1.570796, 1.758625],accel_mss,speed_ms,0,blend_radius_m)
    movel([0.187395, -1.358305, -2.591160, -0.762923, 1.570796, 1.758192],accel_mss,speed_ms,0,blend_radius_m)
    movel([0.186675, -1.360513, -2.589671, -0.762204, 1.570796, 1.757471],accel_mss,speed_ms,0,blend_radius_m)
    movel([0.184681, -1.364824, -2.586745, -0.760820, 1.570796, 1.755477],accel_mss,speed_ms,0,blend_radius_m)
    movel([0.184426, -1.365808, -2.586073, -0.760508, 1.570796, 1.755222],accel_mss,speed_ms,0,blend_radius_m)
    movel([0.184522, -1.366670, -2.585483, -0.760235, 1.570796, 1.755318],accel_mss,speed_ms,0,blend_radius_m)
    movel([0.184952, -1.367245, -2.585090, -0.760054, 1.570796, 1.755749],accel_mss,speed_ms,0,blend_radius_m)
    movel([0.185573, -1.367666, -2.584801, -0.759922, 1.570796, 1.756369],accel_mss,speed_ms,0,blend_radius_m)
    movel([0.186234, -1.368059, -2.584532, -0.759799, 1.570796, 1.757031],accel_mss,speed_ms,0,blend_radius_m)
    movel([0.186781, -1.368550, -2.584194, -0.759645, 1.570796, 1.757577],accel_mss,speed_ms,0,blend_radius_m)
    movel([0.187068, -1.369139, -2.583789, -0.759461, 1.570796, 1.757864],accel_mss,speed_ms,0,blend_radius_m)
    movel([0.187169, -1.369835, -2.583310, -0.759244, 1.570796, 1.757965],accel_mss,speed_ms,0,blend_radius_m)
    movel([0.187036, -1.371377, -2.582245, -0.758767, 1.570796, 1.757832],accel_mss,speed_ms,0,blend_radius_m)
    movel([0.186589, -1.373650, -2.580670, -0.758069, 1.570796, 1.757385],accel_mss,speed_ms,0,blend_radius_m)
    movel([0.185987, -1.375946, -2.579072, -0.757371, 1.570796, 1.756784],accel_mss,speed_ms,0,blend_radius_m)
    movel([0.185230, -1.378254, -2.577458, -0.756677, 1.570796, 1.756026],accel_mss,speed_ms,0,blend_radius_m)
    movel([0.184326, -1.380568, -2.575831, -0.755990, 1.570796, 1.755122],accel_mss,speed_ms,0,blend_radius_m)
    movel([0.183277, -1.382875, -2.574202, -0.755312, 1.570796, 1.754074],accel_mss,speed_ms,0,blend_radius_m)
    movel([0.182094, -1.385167, -2.572576, -0.754646, 1.570796, 1.752890],accel_mss,speed_ms,0,blend_radius_m)
    movel([0.180773, -1.387436, -2.570959, -0.753994, 1.570796, 1.751569],accel_mss,speed_ms,0,blend_radius_m)
    movel([0.179324, -1.389675, -2.569356, -0.753358, 1.570796, 1.750120],accel_mss,speed_ms,0,blend_radius_m)
    movel([0.178313, -1.391062, -2.568359, -0.752968, 1.570796, 1.749109],accel_mss,speed_ms,0,blend_radius_m)
    movel([0.177152, -1.392381, -2.567408, -0.752599, 1.570796, 1.747948],accel_mss,speed_ms,0,blend_radius_m)
    movel([0.175835, -1.393509, -2.566594, -0.752286, 1.570796, 1.746631],accel_mss,speed_ms,0,blend_radius_m)
    movel([0.175117, -1.393958, -2.566269, -0.752162, 1.570796, 1.745913],accel_mss,speed_ms,0,blend_radius_m)
    movel([0.174357, -1.394314, -2.566011, -0.752064, 1.570796, 1.745153],accel_mss,speed_ms,0,blend_radius_m)
    speed_ms = 0.005
    movel([0.174357, -1.385632, -2.562079, -0.764678, 1.570796, 1.745153],accel_mss,speed_ms,0,blend_radius_m)
    speed_ms = 0.040
    movel([0.170630, -1.389375, -2.559393, -0.763621, 1.570796, 1.741426],accel_mss,speed_ms,0,blend_radius_m)
    speed_ms = 0.005
    movel([0.170630, -1.398030, -2.563309, -0.751050, 1.570796, 1.741426],accel_mss,speed_ms,0,blend_radius_m)
    speed_ms = 0.025
    movel([0.170821, -1.398427, -2.563019, -0.750943, 1.570796, 1.741617],accel_mss,speed_ms,0,blend_radius_m)
    movel([0.170755, -1.398945, -2.562640, -0.750804, 1.570796, 1.741551],accel_mss,speed_ms,0,blend_radius_m)
    movel([0.170485, -1.399507, -2.562229, -0.750653, 1.570796, 1.741281],accel_mss,speed_ms,0,blend_radius_m)
    movel([0.170056, -1.400031, -2.561845, -0.750513, 1.570796, 1.740853],accel_mss,speed_ms,0,blend_radius_m)
    movel([0.169408, -1.400513, -2.561492, -0.750384, 1.570796, 1.740205],accel_mss,speed_ms,0,blend_radius_m)
    movel([0.168716, -1.400854, -2.561242, -0.750293, 1.570796, 1.739512],accel_mss,speed_ms,0,blend_radius_m)
    movel([0.168034, -1.401166, -2.561012, -0.750210, 1.570796, 1.738830],accel_mss,speed_ms,0,blend_radius_m)
    movel([0.167427, -1.401563, -2.560721, -0.750105, 1.570796, 1.738223],accel_mss,speed_ms,0,blend_radius_m)
    movel([0.166850, -1.402343, -2.560147, -0.749899, 1.570796, 1.737646],accel_mss,speed_ms,0,blend_radius_m)
    movel([0.166594, -1.402759, -2.559841, -0.749789, 1.570796, 1.737390],accel_mss,speed_ms,0,blend_radius_m)
    movel([0.166221, -1.403177, -2.559532, -0.749679, 1.570796, 1.737017],accel_mss,speed_ms,0,blend_radius_m)
    movel([0.164994, -1.404146, -2.558817, -0.749426, 1.570796, 1.735790],accel_mss,speed_ms,0,blend_radius_m)
    movel([0.163720, -1.404929, -2.558238, -0.749222, 1.570796, 1.734517],accel_mss,speed_ms,0,blend_radius_m)
    movel([0.162395, -1.405553, -2.557776, -0.749060, 1.570796, 1.733191],accel_mss,speed_ms,0,blend_radius_m)
    movel([0.161012, -1.406051, -2.557407, -0.748931, 1.570796, 1.731809],accel_mss,speed_ms,0,blend_radius_m)
    movel([0.161724, -1.405729, -2.557646, -0.749014, 1.570796, 1.732520],accel_mss,speed_ms,0,blend_radius_m)
    movel([0.162436, -1.405503, -2.557813, -0.749073, 1.570796, 1.733233],accel_mss,speed_ms,0,blend_radius_m)
    movel([0.163101, -1.405486, -2.557825, -0.749077, 1.570796, 1.733897],accel_mss,speed_ms,0,blend_radius_m)
    movel([0.163555, -1.405762, -2.557621, -0.749006, 1.570796, 1.734351],accel_mss,speed_ms,0,blend_radius_m)
    movel([0.163626, -1.406299, -2.557223, -0.748867, 1.570796, 1.734423],accel_mss,speed_ms,0,blend_radius_m)
    movel([0.163371, -1.406921, -2.556761, -0.748707, 1.570796, 1.734167],accel_mss,speed_ms,0,blend_radius_m)
    movel([0.162892, -1.407501, -2.556330, -0.748558, 1.570796, 1.733688],accel_mss,speed_ms,0,blend_radius_m)
    movel([0.161307, -1.408781, -2.555377, -0.748232, 1.570796, 1.732103],accel_mss,speed_ms,0,blend_radius_m)
    movel([0.160250, -1.409448, -2.554878, -0.748062, 1.570796, 1.731046],accel_mss,speed_ms,0,blend_radius_m)
    movel([0.159159, -1.410014, -2.554456, -0.747919, 1.570796, 1.729956],accel_mss,speed_ms,0,blend_radius_m)
    movel([0.158046, -1.410469, -2.554116, -0.747805, 1.570796, 1.728842],accel_mss,speed_ms,0,blend_radius_m)
    movel([0.159323, -1.410106, -2.554387, -0.747896, 1.570796, 1.730119],accel_mss,speed_ms,0,blend_radius_m)
    movel([0.160642, -1.409591, -2.554772, -0.748026, 1.570796, 1.731438],accel_mss,speed_ms,0,blend_radius_m)
    movel([0.161935, -1.409111, -2.555130, -0.748148, 1.570796, 1.732731],accel_mss,speed_ms,0,blend_radius_m)
    movel([0.163133, -1.408844, -2.555330, -0.748216, 1.570796, 1.733930],accel_mss,speed_ms,0,blend_radius_m)
    movel([0.163477, -1.408899, -2.555289, -0.748202, 1.570796, 1.734273],accel_mss,speed_ms,0,blend_radius_m)
    movel([0.163505, -1.409116, -2.555126, -0.748146, 1.570796, 1.734302],accel_mss,speed_ms,0,blend_radius_m)
    movel([0.162904, -1.410108, -2.554385, -0.747895, 1.570796, 1.733700],accel_mss,speed_ms,0,blend_radius_m)
    movel([0.162323, -1.410797, -2.553870, -0.747722, 1.570796, 1.733120],accel_mss,speed_ms,0,blend_radius_m)
    movel([0.161658, -1.411434, -2.553393, -0.747562, 1.570796, 1.732455],accel_mss,speed_ms,0,blend_radius_m)
    movel([0.160926, -1.412002, -2.552966, -0.747420, 1.570796, 1.731722],accel_mss,speed_ms,0,blend_radius_m)
    movel([0.161306, -1.411803, -2.553116, -0.747470, 1.570796, 1.732103],accel_mss,speed_ms,0,blend_radius_m)
    movel([0.161741, -1.411686, -2.553204, -0.747499, 1.570796, 1.732537],accel_mss,speed_ms,0,blend_radius_m)
    movel([0.162708, -1.411663, -2.553221, -0.747505, 1.570796, 1.733504],accel_mss,speed_ms,0,blend_radius_m)
    movel([0.163691, -1.411878, -2.553060, -0.747451, 1.570796, 1.734487],accel_mss,speed_ms,0,blend_radius_m)
    movel([0.164559, -1.412269, -2.552766, -0.747354, 1.570796, 1.735355],accel_mss,speed_ms,0,blend_radius_m)
    movel([0.165183, -1.412777, -2.552384, -0.747228, 1.570796, 1.735979],accel_mss,speed_ms,0,blend_radius_m)
    movel([0.165433, -1.413340, -2.551961, -0.747088, 1.570796, 1.736229],accel_mss,speed_ms,0,blend_radius_m)
    movel([0.165377, -1.413622, -2.551748, -0.747018, 1.570796, 1.736173],accel_mss,speed_ms,0,blend_radius_m)
    movel([0.165178, -1.413895, -2.551543, -0.746951, 1.570796, 1.735975],accel_mss,speed_ms,0,blend_radius_m)
    movel([0.164824, -1.414153, -2.551349, -0.746887, 1.570796, 1.735620],accel_mss,speed_ms,0,blend_radius_m)
    movel([0.164293, -1.414386, -2.551173, -0.746830, 1.570796, 1.735089],accel_mss,speed_ms,0,blend_radius_m)
    movel([0.163692, -1.414504, -2.551084, -0.746801, 1.570796, 1.734488],accel_mss,speed_ms,0,blend_radius_m)
    movel([0.161386, -1.414269, -2.551261, -0.746859, 1.570796, 1.732182],accel_mss,speed_ms,0,blend_radius_m)
    movel([0.160491, -1.414222, -2.551297, -0.746870, 1.570796, 1.731287],accel_mss,speed_ms,0,blend_radius_m)
    movel([0.159544, -1.414322, -2.551221, -0.746846, 1.570796, 1.730340],accel_mss,speed_ms,0,blend_radius_m)
    movel([0.157916, -1.414850, -2.550823, -0.746716, 1.570796, 1.728713],accel_mss,speed_ms,0,blend_radius_m)
    movel([0.156281, -1.415480, -2.550347, -0.746562, 1.570796, 1.727077],accel_mss,speed_ms,0,blend_radius_m)
    movel([0.155455, -1.415677, -2.550198, -0.746514, 1.570796, 1.726251],accel_mss,speed_ms,0,blend_radius_m)
    movel([0.154674, -1.415717, -2.550168, -0.746504, 1.570796, 1.725470],accel_mss,speed_ms,0,blend_radius_m)
    movel([0.154031, -1.415553, -2.550292, -0.746544, 1.570796, 1.724828],accel_mss,speed_ms,0,blend_radius_m)
    movel([0.153621, -1.415146, -2.550600, -0.746644, 1.570796, 1.724417],accel_mss,speed_ms,0,blend_radius_m)
    movel([0.154382, -1.414371, -2.551185, -0.746834, 1.570796, 1.725178],accel_mss,speed_ms,0,blend_radius_m)
    movel([0.155220, -1.413659, -2.551721, -0.747009, 1.570796, 1.726016],accel_mss,speed_ms,0,blend_radius_m)
    speed_ms = 0.005
    movel([0.155220, -1.405120, -2.547873, -0.759396, 1.570796, 1.726016],accel_mss,speed_ms,0,blend_radius_m)
    speed_ms = 0.040
    movel([0.163508, -1.410385, -2.543940, -0.758065, 1.570796, 1.734304],accel_mss,speed_ms,0,blend_radius_m)
    speed_ms = 0.005
    movel([0.163508, -1.418884, -2.547766, -0.745739, 1.570796, 1.734304],accel_mss,speed_ms,0,blend_radius_m)
    speed_ms = 0.025
    movel([0.164040, -1.418327, -2.548189, -0.745873, 1.570796, 1.734837],accel_mss,speed_ms,0,blend_radius_m)
    movel([0.164735, -1.417965, -2.548464, -0.745960, 1.570796, 1.735532],accel_mss,speed_ms,0,blend_radius_m)
    movel([0.165471, -1.417814, -2.548579, -0.745996, 1.570796, 1.736267],accel_mss,speed_ms,0,blend_radius_m)
    movel([0.166119, -1.417892, -2.548520, -0.745977, 1.570796, 1.736915],accel_mss,speed_ms,0,blend_radius_m)
    movel([0.166608, -1.418166, -2.548311, -0.745911, 1.570796, 1.737404],accel_mss,speed_ms,0,blend_radius_m)
    movel([0.166973, -1.418561, -2.548011, -0.745817, 1.570796, 1.737770],accel_mss,speed_ms,0,blend_radius_m)
    movel([0.167483, -1.419534, -2.547271, -0.745584, 1.570796, 1.738279],accel_mss,speed_ms,0,blend_radius_m)
    movel([0.167928, -1.418810, -2.547822, -0.745757, 1.570796, 1.738724],accel_mss,speed_ms,0,blend_radius_m)
    movel([0.168163, -1.418075, -2.548381, -0.745933, 1.570796, 1.738960],accel_mss,speed_ms,0,blend_radius_m)
    movel([0.168172, -1.417391, -2.548900, -0.746098, 1.570796, 1.738968],accel_mss,speed_ms,0,blend_radius_m)
    movel([0.167947, -1.416813, -2.549338, -0.746238, 1.570796, 1.738743],accel_mss,speed_ms,0,blend_radius_m)
    movel([0.168394, -1.417058, -2.549153, -0.746179, 1.570796, 1.739190],accel_mss,speed_ms,0,blend_radius_m)
    movel([0.168736, -1.417394, -2.548898, -0.746097, 1.570796, 1.739532],accel_mss,speed_ms,0,blend_radius_m)
    movel([0.169157, -1.418275, -2.548229, -0.745885, 1.570796, 1.739954],accel_mss,speed_ms,0,blend_radius_m)
    movel([0.169328, -1.419332, -2.547425, -0.745632, 1.570796, 1.740125],accel_mss,speed_ms,0,blend_radius_m)
    movel([0.169353, -1.420450, -2.546572, -0.745367, 1.570796, 1.740149],accel_mss,speed_ms,0,blend_radius_m)
    movel([0.169176, -1.421714, -2.545607, -0.745069, 1.570796, 1.739972],accel_mss,speed_ms,0,blend_radius_m)
    movel([0.168797, -1.422936, -2.544671, -0.744783, 1.570796, 1.739594],accel_mss,speed_ms,0,blend_radius_m)
    movel([0.168392, -1.424137, -2.543748, -0.744504, 1.570796, 1.739189],accel_mss,speed_ms,0,blend_radius_m)
    movel([0.168132, -1.425343, -2.542820, -0.744226, 1.570796, 1.738928],accel_mss,speed_ms,0,blend_radius_m)
    movel([0.167512, -1.424656, -2.543349, -0.744384, 1.570796, 1.738308],accel_mss,speed_ms,0,blend_radius_m)
    movel([0.166680, -1.424178, -2.543716, -0.744494, 1.570796, 1.737476],accel_mss,speed_ms,0,blend_radius_m)
    movel([0.165663, -1.423940, -2.543899, -0.744549, 1.570796, 1.736459],accel_mss,speed_ms,0,blend_radius_m)
    movel([0.164483, -1.423974, -2.543874, -0.744542, 1.570796, 1.735279],accel_mss,speed_ms,0,blend_radius_m)
    speed_ms = 0.005
    movel([0.164483, -1.415513, -2.540069, -0.756806, 1.570796, 1.735279],accel_mss,speed_ms,0,blend_radius_m)
    speed_ms = 0.040
    movel([0.165977, -1.419219, -2.537249, -0.755922, 1.570796, 1.736773],accel_mss,speed_ms,0,blend_radius_m)
    speed_ms = 0.005
    movel([0.165977, -1.427651, -2.541037, -0.743700, 1.570796, 1.736773],accel_mss,speed_ms,0,blend_radius_m)
    speed_ms = 0.025
    movel([0.166267, -1.429145, -2.539879, -0.743365, 1.570796, 1.737064],accel_mss,speed_ms,0,blend_radius_m)
    movel([0.166820, -1.430497, -2.538828, -0.743064, 1.570796, 1.737617],accel_mss,speed_ms,0,blend_radius_m)
    movel([0.167712, -1.431570, -2.537993, -0.742827, 1.570796, 1.738509],accel_mss,speed_ms,0,blend_radius_m)
    movel([0.168312, -1.431959, -2.537689, -0.742741, 1.570796, 1.739108],accel_mss,speed_ms,0,blend_radius_m)
    movel([0.169029, -1.432228, -2.537479, -0.742682, 1.570796, 1.739825],accel_mss,speed_ms,0,blend_radius_m)
    movel([0.170162, -1.432372, -2.537366, -0.742651, 1.570796, 1.740959],accel_mss,speed_ms,0,blend_radius_m)
    movel([0.171382, -1.432282, -2.537437, -0.742671, 1.570796, 1.742178],accel_mss,speed_ms,0,blend_radius_m)
    movel([0.172671, -1.432011, -2.537648, -0.742730, 1.570796, 1.743467],accel_mss,speed_ms,0,blend_radius_m)
    movel([0.174010, -1.431616, -2.537957, -0.742817, 1.570796, 1.744807],accel_mss,speed_ms,0,blend_radius_m)
    movel([0.176764, -1.430663, -2.538699, -0.743027, 1.570796, 1.747560],accel_mss,speed_ms,0,blend_radius_m)
    movel([0.179491, -1.429863, -2.539322, -0.743204, 1.570796, 1.750287],accel_mss,speed_ms,0,blend_radius_m)
    movel([0.181013, -1.429635, -2.539499, -0.743255, 1.570796, 1.751809],accel_mss,speed_ms,0,blend_radius_m)
    movel([0.182461, -1.429621, -2.539510, -0.743258, 1.570796, 1.753257],accel_mss,speed_ms,0,blend_radius_m)
    movel([0.183810, -1.429810, -2.539363, -0.743216, 1.570796, 1.754607],accel_mss,speed_ms,0,blend_radius_m)
    movel([0.185034, -1.430194, -2.539064, -0.743131, 1.570796, 1.755830],accel_mss,speed_ms,0,blend_radius_m)
    movel([0.186110, -1.430760, -2.538624, -0.743005, 1.570796, 1.756906],accel_mss,speed_ms,0,blend_radius_m)
    movel([0.187012, -1.431499, -2.538048, -0.742842, 1.570796, 1.757809],accel_mss,speed_ms,0,blend_radius_m)
    movel([0.187715, -1.432399, -2.537345, -0.742645, 1.570796, 1.758511],accel_mss,speed_ms,0,blend_radius_m)
    movel([0.188198, -1.433447, -2.536525, -0.742416, 1.570796, 1.758995],accel_mss,speed_ms,0,blend_radius_m)
    speed_ms = 0.005
    movel([0.188198, -1.425059, -2.532761, -0.754569, 1.570796, 1.758995],accel_mss,speed_ms,0,blend_radius_m)
    speed_ms = 0.040
    movel([0.160347, -1.408053, -2.545687, -0.758649, 1.570796, 1.731144],accel_mss,speed_ms,0,blend_radius_m)
    speed_ms = 0.005
    movel([0.160347, -1.416570, -2.549523, -0.746297, 1.570796, 1.731144],accel_mss,speed_ms,0,blend_radius_m)
    speed_ms = 0.025
    movel([0.161048, -1.416837, -2.549320, -0.746232, 1.570796, 1.731844],accel_mss,speed_ms,0,blend_radius_m)
    movel([0.161576, -1.417274, -2.548989, -0.746126, 1.570796, 1.732372],accel_mss,speed_ms,0,blend_radius_m)
    movel([0.161701, -1.417602, -2.548740, -0.746047, 1.570796, 1.732497],accel_mss,speed_ms,0,blend_radius_m)
    movel([0.161690, -1.417989, -2.548446, -0.745954, 1.570796, 1.732487],accel_mss,speed_ms,0,blend_radius_m)
    movel([0.161538, -1.418393, -2.548139, -0.745857, 1.570796, 1.732334],accel_mss,speed_ms,0,blend_radius_m)
    movel([0.161230, -1.418767, -2.547855, -0.745767, 1.570796, 1.732027],accel_mss,speed_ms,0,blend_radius_m)
    movel([0.160492, -1.419336, -2.547422, -0.745631, 1.570796, 1.731288],accel_mss,speed_ms,0,blend_radius_m)
    movel([0.160242, -1.419699, -2.547145, -0.745545, 1.570796, 1.731038],accel_mss,speed_ms,0,blend_radius_m)
    movel([0.160152, -1.420075, -2.546859, -0.745456, 1.570796, 1.730949],accel_mss,speed_ms,0,blend_radius_m)
    movel([0.160302, -1.420762, -2.546335, -0.745293, 1.570796, 1.731098],accel_mss,speed_ms,0,blend_radius_m)
    movel([0.160720, -1.421423, -2.545829, -0.745137, 1.570796, 1.731517],accel_mss,speed_ms,0,blend_radius_m)
    movel([0.161277, -1.421975, -2.545406, -0.745007, 1.570796, 1.732073],accel_mss,speed_ms,0,blend_radius_m)
    movel([0.161958, -1.422414, -2.545071, -0.744905, 1.570796, 1.732754],accel_mss,speed_ms,0,blend_radius_m)
    movel([0.162749, -1.422724, -2.544833, -0.744832, 1.570796, 1.733545],accel_mss,speed_ms,0,blend_radius_m)
    movel([0.162178, -1.423539, -2.544208, -0.744642, 1.570796, 1.732975],accel_mss,speed_ms,0,blend_radius_m)
    movel([0.161765, -1.424363, -2.543574, -0.744451, 1.570796, 1.732562],accel_mss,speed_ms,0,blend_radius_m)
    movel([0.161491, -1.425192, -2.542936, -0.744261, 1.570796, 1.732287],accel_mss,speed_ms,0,blend_radius_m)
    movel([0.161335, -1.426018, -2.542300, -0.744072, 1.570796, 1.732131],accel_mss,speed_ms,0,blend_radius_m)
    movel([0.161310, -1.427628, -2.541056, -0.743706, 1.570796, 1.732106],accel_mss,speed_ms,0,blend_radius_m)
    movel([0.161552, -1.429136, -2.539887, -0.743367, 1.570796, 1.732348],accel_mss,speed_ms,0,blend_radius_m)
    movel([0.161818, -1.430578, -2.538765, -0.743046, 1.570796, 1.732614],accel_mss,speed_ms,0,blend_radius_m)
    movel([0.161818, -1.431340, -2.538172, -0.742877, 1.570796, 1.732614],accel_mss,speed_ms,0,blend_radius_m)
    movel([0.161643, -1.432142, -2.537546, -0.742701, 1.570796, 1.732440],accel_mss,speed_ms,0,blend_radius_m)
    movel([0.161209, -1.432975, -2.536895, -0.742519, 1.570796, 1.732006],accel_mss,speed_ms,0,blend_radius_m)
    movel([0.160534, -1.433740, -2.536296, -0.742353, 1.570796, 1.731330],accel_mss,speed_ms,0,blend_radius_m)
    movel([0.159706, -1.434315, -2.535846, -0.742229, 1.570796, 1.730503],accel_mss,speed_ms,0,blend_radius_m)
    movel([0.158821, -1.434572, -2.535644, -0.742173, 1.570796, 1.729617],accel_mss,speed_ms,0,blend_radius_m)
    movel([0.159210, -1.435121, -2.535213, -0.742055, 1.570796, 1.730006],accel_mss,speed_ms,0,blend_radius_m)
    movel([0.159647, -1.436428, -2.534185, -0.741776, 1.570796, 1.730443],accel_mss,speed_ms,0,blend_radius_m)
    movel([0.159693, -1.437162, -2.533607, -0.741620, 1.570796, 1.730489],accel_mss,speed_ms,0,blend_radius_m)
    movel([0.159449, -1.438725, -2.532372, -0.741291, 1.570796, 1.730245],accel_mss,speed_ms,0,blend_radius_m)
    movel([0.159158, -1.439530, -2.531736, -0.741124, 1.570796, 1.729954],accel_mss,speed_ms,0,blend_radius_m)
    movel([0.158753, -1.440335, -2.531097, -0.740957, 1.570796, 1.729550],accel_mss,speed_ms,0,blend_radius_m)
    speed_ms = 0.005
    movel([0.158753, -1.432000, -2.527362, -0.753027, 1.570796, 1.729550],accel_mss,speed_ms,0,blend_radius_m)
    speed_ms = 0.040
    movel([0.154357, -1.432582, -2.526906, -0.752901, 1.570796, 1.725154],accel_mss,speed_ms,0,blend_radius_m)
    speed_ms = 0.005
    movel([0.154357, -1.440913, -2.530638, -0.740838, 1.570796, 1.725154],accel_mss,speed_ms,0,blend_radius_m)
    speed_ms = 0.025
    movel([0.157061, -1.447582, -2.525307, -0.739499, 1.570796, 1.727858],accel_mss,speed_ms,0,blend_radius_m)
    movel([0.157277, -1.448453, -2.524606, -0.739330, 1.570796, 1.728073],accel_mss,speed_ms,0,blend_radius_m)
    movel([0.157213, -1.448926, -2.524225, -0.739238, 1.570796, 1.728009],accel_mss,speed_ms,0,blend_radius_m)
    movel([0.156951, -1.449404, -2.523839, -0.739146, 1.570796, 1.727748],accel_mss,speed_ms,0,blend_radius_m)
    movel([0.156049, -1.450346, -2.523078, -0.738965, 1.570796, 1.726845],accel_mss,speed_ms,0,blend_radius_m)
    movel([0.155895, -1.450870, -2.522654, -0.738865, 1.570796, 1.726691],accel_mss,speed_ms,0,blend_radius_m)
    movel([0.155988, -1.451343, -2.522271, -0.738775, 1.570796, 1.726784],accel_mss,speed_ms,0,blend_radius_m)
    movel([0.156429, -1.451974, -2.521759, -0.738655, 1.570796, 1.727225],accel_mss,speed_ms,0,blend_radius_m)
    movel([0.157105, -1.452459, -2.521366, -0.738564, 1.570796, 1.727901],accel_mss,speed_ms,0,blend_radius_m)
